fbPulseCtrl[1].Q;
fbPulseCtrl[1].RT;
fbPulseCtrl[2].Q;
fbPulseCtrl[2].RT;
fbPulseCtrl[3].Q;
fbPulseCtrl[3].RT;
fbPulseCtrl[4].Q;
fbPulseCtrl[4].RT;
fbPulseCtrl[5].Q;
fbPulseCtrl[5].RT;
fbPulseCtrl[6].Q;
fbPulseCtrl[6].RT;
fbPulseCtrl[7].Q;
fbPulseCtrl[7].RT;
fbPulseCtrl[8].Q;
fbPulseCtrl[8].RT;


IF bWaterOn AND ( bWaterOn2   OR    ABS( arrAxisCtrl[P1AxisNo.GMWind_U].Status.fActVelo)>=5 AND  ABS (arrAxisCtrl[P1AxisNo.GMWind_D].Status.fActVelo)>=5 )   THEN
  //P3EL2889S[3,5]:= fbPulseCtrl[9].Q;
   P1EL2889S[3,1]:= fbPulseCtrl[9].Q;
   P1EL2889S[3,2]:= fbPulseCtrl[9].Q;

   P2EL2889S[4,1]:=fbPulseCtrl[9].Q	;	
   P2EL2889S[4,2]:=fbPulseCtrl[9].Q;	

   P2EL2889S[4,3]:=fbPulseCtrl[9].Q	;	
   P2EL2889S[4,4]:=fbPulseCtrl[9].Q;	

ELSE
  //P3EL2889S[3,5]:= FALSE;
   P1EL2889S[3,1]:= FALSE;
   P1EL2889S[3,2]:= FALSE;
   P2EL2889S[4,1]:= FALSE	;	
   P2EL2889S[4,2]:= FALSE;	

   P2EL2889S[4,3]:=FALSE	;	
   P2EL2889S[4,4]:=FALSE;	
END_IF


//P1EL2889S[3,1]


*)
END_ACTION

ACTION TempBasic:


FOR i:=1 TO MaxTemp DO   //显示温度转换
	IF TempPVs[i].iPV1<>9999 THEN
		TempPVs[i].fPV1:=TempPVs[i].iPV1/10;	
	ELSE
		TempPVs[i].fPV1:=999.9;
	END_IF
    arrTempCtrl[i].fPVShow1:=TempPVs[i].fPV1;
	
	IF TempPVs[i].iPV2<>9999 THEN
		TempPVs[i].fPV2:=TempPVs[i].iPV2/10;
	ELSE
		TempPVs[i].fPV2:=999.9;
	END_IF
	 arrTempCtrl[i].fPVShow2:=TempPVs[i].fPV2;

	IF TempPVs[i].iPV3<>9999 THEN
		TempPVs[i].fPV3:=TempPVs[i].iPV3/10;
	ELSE
		TempPVs[i].fPV3:=999.9;
	END_IF
	 arrTempCtrl[i].fPVShow3:=TempPVs[i].fPV3;

	IF TempPVs[i].iPV4<>9999 THEN
		TempPVs[i].fPV4:=TempPVs[i].iPV4/10;
	ELSE
		TempPVs[i].fPV4:=999.9;
	END_IF
    arrTempCtrl[i].fPVShow4:=TempPVs[i].fPV4;
END_FOR

//温度控制
FOR i:=1 TO MaxTemp DO
     fbTemp[i](bReset:=P3_SystemRUN.bReset , ParTemp:=arrTempPar[i] , TempCtrl:=arrTempCtrl[i] );
END_FOR
END_ACTION

END_PROGRAM

// ---- P3POUs/P3FB/FB_Temperature.TcPOU
FUNCTION_BLOCK FB_Temperature    //温控功能块
VAR_INPUT
    bReset          :BOOL;
	ParTemp      : ST_ParTemperature;
END_VAR

VAR_IN_OUT
     TempCtrl:     STTempCtrl;
END_VAR
VAR_OUTPUT
    
END_VAR




VAR
       fTempMax                                :REAL;     //温度上限
      fTempMin                                 :REAL;     //温度下限


       rtTemp  :ARRAY[1..4] OF Tc2_Standard.R_TRIG;
	  iCountShow: INT;  //使用的显示通道数量
	  TemTON :Tc2_Standard.TON;
END_VAR

ParTemp.fTempArea:=5;
TemTON(PT:=T#300S);

TempCtrl.Tem_fPV:=TempCtrl.In.fPV-ParTemp.Tem_Offset;
TempCtrl.fPVShow_1:=TempCtrl.fPVShow1-ParTemp.Tem_Offset;
TempCtrl.In.fPV:=TempCtrl.In.iPV/10; //当前温度显示

TempCtrl.Out.iSV:=           REAL_TO_INT(ParTemp.fTempSet+ParTemp.Tem_Offset)*10; //控制温度设定值
//TempCtrl.Out.iPV_Offset:= REAL_TO_INT(ParTemp.fTempSet)*10;//控制温度设定值

//启动加热时候   如果当前温度到达设定温度 范围内则开始 判断温度超温和低温报警     
//启动加热5分钟  当前温度还未到达设定温度范围  则报警低温报警
//控制温度和显示温度实时检测差值并判断报警


(**自整定报警**)
TempCtrl.bTuningError:=TempCtrl.In.AutoTuningerr;  //
(**超温报警**)
//IF TempCtrl.In.AutoTuningON OR TempCtrl.In.HeatingON THEN
      rtTemp[1](CLK:=TempCtrl.Tem_fPV>ParTemp.fTempMax , Q=> );  //超温报警
      IF  (*rtTemp[1].Q*) TempCtrl.Tem_fPV>ParTemp.fTempMax+5 OR TempCtrl.fPVShow_1 >ParTemp.fTempMax+10 THEN
          TempCtrl.bTempError_HI:=TRUE;
      END_IF
//END_IF


(**传感器检测异常报警**)
  iCountShow:=SEL(TempCtrl.fPVShow_1<>999.9, 0,1)+SEL(TempCtrl.fPVShow2<>999.9, 0,1) +SEL(TempCtrl.fPVShow3<>999.9, 0,1) + SEL(TempCtrl.fPVShow4<>999.9, 0,1) ;

CASE  iCountShow OF 
1:
IF TempCtrl.In.PIDON AND  ABS (ParTemp.fTempSet-TempCtrl.Tem_fPV)<ParTemp.fTempArea AND NOT TempCtrl.bSenserError AND NOT TempCtrl.bTempError_HI  THEN
	iCountShow:=10;
END_IF

 
 
10:
    
      rtTemp[2](CLK:=ABS (TempCtrl.Tem_fPV-TempCtrl.fPVShow_1)>=ParTemp.fTempArea , Q=> );  //超温报警
       IF ABS (TempCtrl.Tem_fPV-TempCtrl.fPVShow_1)>=ParTemp.fTempArea THEN
             TempCtrl.bSenserError:=TRUE;
      END_IF
	  IF NOT TempCtrl.In.PIDON THEN
		  iCountShow:=0;
	  END_IF
	  
(*2:
      rtTemp[2](CLK:=ABS (TempCtrl.In.fPV-TempCtrl.fPVShow1)>=ParTemp.fTempArea  OR   
                              ABS (TempCtrl.In.fPV-TempCtrl.fPVShow2)>=ParTemp.fTempArea, Q=> );  //超温报警
       IF rtTemp[2].Q THEN
             TempCtrl.bSenserError:=TRUE;
      END_IF
3:
      rtTemp[2](CLK:=ABS (TempCtrl.In.fPV-TempCtrl.fPVShow1)>=ParTemp.fTempArea  OR   
                              ABS (TempCtrl.In.fPV-TempCtrl.fPVShow2)>=ParTemp.fTempArea  OR   
                              ABS (TempCtrl.In.fPV-TempCtrl.fPVShow3)>=ParTemp.fTempArea, Q=> );  //超温报警
       IF rtTemp[2].Q THEN
             TempCtrl.bSenserError:=TRUE;
      END_IF
4:
      rtTemp[2](CLK:=ABS (TempCtrl.In.fPV-TempCtrl.fPVShow1)>=ParTemp.fTempArea  OR   
                              ABS (TempCtrl.In.fPV-TempCtrl.fPVShow2)>=ParTemp.fTempArea  OR   
                              ABS (TempCtrl.In.fPV-TempCtrl.fPVShow3)>=ParTemp.fTempArea  OR   
                              ABS (TempCtrl.In.fPV-TempCtrl.fPVShow4)>=ParTemp.fTempArea, Q=> );  //超温报警
       IF rtTemp[2].Q THEN
             TempCtrl.bSenserError:=TRUE;
      END_IF*)
END_CASE

 IF TempCtrl.In.PIDON AND ABS (ParTemp.fTempSet-TempCtrl.Tem_fPV)>=ParTemp.fTempArea THEN
	 TemTON.IN:=TRUE;
	 ELSE
    TemTON.IN:=FALSE;	 
 END_IF
IF TemTON.Q THEN
	TempCtrl.bTempError_LI:=TRUE;
END_IF

IF bReset AND ( TempCtrl.bTempError_HI OR TempCtrl.bSenserError OR TempCtrl.bTempError_LI ) THEN
    TempCtrl.bTempError_HI:=FALSE;
    TempCtrl.bSenserError:=FALSE;
	TempCtrl.bTempError_LI:=FALSE;
END_IF


IF TempCtrl.bTempError_HI OR TempCtrl.bSenserError OR TempCtrl.bTempError_LI THEN
	TempCtrl.Out.PIDRun:=FALSE;
END_IF















(*
rtRec[1](CLK:=RecCtrl.Cmd.bLock , Q=> );
rtRec[2](CLK:=RecCtrl.Cmd.bAuto , Q=> );
rtRec[3](CLK:=RecCtrl.Cmd.bManual , Q=> );
rtRec[4](CLK:=RecCtrl.Cmd.bCentre , Q=> );

IF rtRec[1].Q   THEN  //外部锁定
    RecCtrl.Io.boLock:=TRUE;
    RecCtrl.Io.boAuto:=FALSE;
    RecCtrl.Io.boManual:=FALSE;
    RecCtrl.Io.boCentre:=FALSE;
END_IF

IF rtRec[2].Q   THEN  //自动
    RecCtrl.Io.boLock:=FALSE;
    RecCtrl.Io.boAuto:=TRUE;
    RecCtrl.Io.boManual:=FALSE;
    RecCtrl.Io.boCentre:=FALSE;
END_IF

IF rtRec[3].Q   THEN  //手动
    RecCtrl.Io.boLock:=FALSE;
    RecCtrl.Io.boAuto:=FALSE;
    RecCtrl.Io.boManual:=TRUE;
    RecCtrl.Io.boCentre:=FALSE;
END_IF

IF rtRec[4].Q   THEN  //居中
    RecCtrl.Io.boLock:=FALSE;
    RecCtrl.Io.boAuto:=FALSE;
    RecCtrl.Io.boManual:=FALSE;
    RecCtrl.Io.boCentre:=TRUE;
END_IF


RecCtrl.Status.bError:=RecCtrl.Io.biError;
RecCtrl.Status.bRuning:=RecCtrl.Io.biCentre;


*)

END_FUNCTION_BLOCK

// ---- P3POUs/POUs/Auxiliary/LateBlanking_Alarm.TcPOU
PROGRAM LateBlanking_Alarm
VAR
	Twinkle :ARRAY[1..20] OF FB_Blink;
	FB_Blink_11: FB_Blink;
	Alarm_TON :ARRAY[1..100] OF Tc2_Standard.TON;
	 AxisHandautomatic1: FB_AxisHandautomatic_1;
	 rAlarm :ARRAY[1..10] OF R_TRIG;
	 CleanTrig: R_TRIG;
END_VAR

QY_error:=YL_I[1];
Alarm();

Alarm_TON[1](PT:=T#5S);
Alarm_TON[2](PT:=T#5S);
Alarm_TON[3](PT:=T#5S);
Alarm_TON[4](PT:=T#8S);
Alarm_TON[5](PT:=T#8S);
Alarm_TON[6](PT:=T#10MS);
Alarm_TON[7](PT:=T#10MS);
Alarm_TON[8](PT:=T#10MS);
Alarm_TON[9](PT:=T#10MS);
Alarm_TON[10](PT:=T#10MS);
Alarm_TON[11](PT:=T#10MS);
Alarm_TON[12](PT:=T#10MS);
Alarm_TON[13](PT:=T#10MS);
Alarm_TON[14](PT:=T#10MS);
Alarm_TON[15](PT:=T#100MS);
Alarm_TON[16](PT:=T#100MS);
Alarm_TON[17](PT:=T#100MS);
Alarm_TON[18](PT:=T#100MS);
Alarm_TON[19](PT:=T#20MS);
Alarm_TON[20](PT:=T#6S);
Alarm_TON[25](PT:=T#60MS);
Alarm_TON[26](PT:=T#60MS);
Alarm_TON[27](PT:=T#200MS);
Alarm_TON[31](PT:=T#1.1S);
Alarm_TON[32](PT:=T#1.1S);
Alarm_TON[33](PT:=T#1.1S);
Alarm_TON[34](PT:=T#1000MS);
Alarm_TON[35](PT:=T#2000MS);
Alarm_TON[36](PT:=T#2S);
Alarm_TON[37](PT:=T#2S);
Alarm_TON[38](PT:=T#60MS);
Alarm_TON[39](PT:=T#60MS);
Alarm_TON[40](PT:=T#3S);
//尾段报警总结
IF  arrAxisCtrl[P3AxisNo.P3M1_ColdpreActuated].Status.Error             OR arrAxisCtrl[P3AxisNo.P3M1_ColdpreLine].Status.Error           OR
	arrAxisCtrl[P3AxisNo.P3M1_ColdpreRetracting].Status.Error           OR arrAxisCtrl[P3AxisNo.P3M1_ColdpreSupPlateLine].Status.Error   OR
	arrAxisCtrl[P3AxisNo.P3M1_ColdpreUpDown].Status.Error               OR arrAxisCtrl[P3AxisNo.P3M1_ColdpreWhirling].Status.Error       OR
	arrAxisCtrlV2[P3AxisNo.P3_M2_OvenCarrying].Status.Error             OR arrAxisCtrlV2[P3AxisNo.P3_M2_OvenRetracting].Status.Error       OR
	arrAxisCtrlV2[P3AxisNo.P3_M2_OvenUpDown].Status.Error               OR arrAxisCtrl[P3AxisNo.P3_M3_HotPressingActuated].Status.Error  OR
	arrAxisCtrl[P3AxisNo.P3_M3_HotPressingLine].Status.Error            OR arrAxisCtrl[P3AxisNo.P3_M4_OffloadingCarrying].Status.Error   OR
	arrAxisCtrl[P3AxisNo.P3_M4_OffloadingUpDown].Status.Error           OR arrAxisCtrl[P3AxisNo.P3_M4_SortingoutCarrying].Status.Error   OR
	//arrAxisCtrl[P3AxisNo.P3_M4_SortingoutUpDown].Status.Error           OR arrAxisCtrl[P3AxisNo.P3_M4_WeighLine].Status.Error            OR
	arrAxisCtrl[P3AxisNo.P3_M4_WeighUpDown].Status.Error                OR arrAxisCtrl[P3AxisNo.P3_M4_WeighWhirling].Status.Error        OR
	//一号叠台、尾卷、贴胶电机报警
	
	(*arrCyCtrl[P3CYNo.P3ColdPressClip].Status.Error1                     OR*) (*arrCyCtrl[P3CYNo.P3ColdPressTensed].Status.Error1             OR
	arrCyCtrl[P3CYNo.P3HotPressTensed].Status.Error1                    OR*arrCyCtrl[P3CYNo.P3OvenMoveClip].Status.Error1           (  OR
	arrCyCtrl[P3CYNo.P3ShortTest].Status.Error1                        OR*)  arrCyCtrl[P3CYNo.P3SortClamp].Status.Error1                   OR
	arrCyCtrl[P3CYNo.P3SortLifting].Status.Error1                       OR arrCyCtrl[P3CYNo.P3SortRotate].Status.Error1                  OR
	arrCyCtrl[P3CYNo.P3ThicknessMeasuringSwitch].Status.Error1          OR arrCyCtrl[P3CYNo.P3ThicknessPressure].Status.Error1           OR
	arrCyCtrl[P3CYNo.P3ThicknessSupport].Status.Error1                  OR arrCyCtrl[P3CYNo.P3WeightFeedingClamp].Status.Error1          OR
	arrCyCtrl[P3CYNo.P3BoxLock1_NG].Status.Error1                       OR arrCyCtrl[P3CYNo.P3BoxLock2_NG].Status.Error1                 OR
	arrCyCtrl[P3CYNo.P3BoxLock3_NG].Status.Error1                       OR arrCyCtrl[P3CYNo.P3BlankingClamp].Status.Error1               OR
	arrCyCtrl[P3CYNo.P3BlankingLifting].Status.Error1                   OR arrCyCtrl[P3CYNo.P3Oven1].Status.Error1                       OR
	arrCyCtrl[P3CYNo.P3Oven2].Status.Error1                             OR arrCyCtrl[P3CYNo.P3Oven3].Status.Error1                       OR
	arrCyCtrl[P3CYNo.P3Oven4].Status.Error1                             OR arrCyCtrl[P3CYNo.P3Oven5].Status.Error1                       OR
	arrCyCtrl[P3CYNo.P3Oven6].Status.Error1                             OR arrCyCtrl[P3CYNo.P3Oven7].Status.Error1                       OR
	arrCyCtrl[P3CYNo.P3Oven8].Status.Error1                             OR arrCyCtrl[P3CYNo.P3Oven9].Status.Error1                       OR
	arrCyCtrl[P3CYNo.P3Oven10].Status.Error1                            OR arrCyCtrl[P3CYNo.P3Oven11].Status.Error1                      OR
	arrCyCtrl[P3CYNo.P3Oven12].Status.Error1                            OR arrCyCtrl[P3CYNo.P3Oven13].Status.Error1                      OR
	arrCyCtrl[P3CYNo.P3Oven14].Status.Error1                            OR arrCyCtrl[P3CYNo.P3Oven15].Status.Error1                      OR
	arrCyCtrl[P3CYNo.P3Oven16].Status.Error1                            OR arrCyCtrl[P3CYNo.P3Oven17].Status.Error1                      OR
	arrCyCtrl[P3CYNo.P3Oven18].Status.Error1                            OR arrCyCtrl[P3CYNo.P3Oven19].Status.Error1                      OR
	arrCyCtrl[P3CYNo.P3Oven20].Status.Error1                            OR arrCyCtrl[P3CYNo.P3Oven21].Status.Error1                      OR
	arrCyCtrl[P3CYNo.P3CellPush].Status.Error1                          OR arrCyCtrl[P3CYNo.P3CellAdvance].Status.Error1                 OR
	arrCyCtrl[P3CYNo.P3TapePush].Status.Error1                          OR arrCyCtrl[P3CYNo.P3TapePull].Status.Error1                    OR
	arrCyCtrl[P3CYNo.P3TapeLift].Status.Error1                          OR arrCyCtrl[P3CYNo.P3TapeCut].Status.Error1                     OR
	arrCyCtrl[P3CYNo.P3GluePush].Status.Error1                          OR arrCyCtrl[P3CYNo.P3TapeBuffer].Status.Error1                  OR
	arrCyCtrl[P3CYNo.P3TapeSpin].Status.Error1                          OR arrCyCtrl[P3CYNo.P3WgightUP].Status.Error1                    OR
	arrCyCtrl[P3CYNo.P3SortPush].Status.Error1                          OR arrCyCtrl[P3CYNo.P3CellPushSpin].Status.Error1                OR
	arrCyCtrl[P3CYNo.P3CellSpin].Status.Error1                          OR arrCyCtrl[P3CYNo.P3_GlueExtend].Status.Error1                 OR
	arrCyCtrl[P3CYNo.P3_GluePress].Status.Error1                        OR arrCyCtrl[P3CYNo.P3_GlueCut].Status.Error1                    OR
	arrCyCtrl[P3CYNo.P3_GluePull].Status.Error1                         OR
    //尾段气缸ON报警
	
	arrCyCtrl[P3CYNo.P3ColdPressClip].Status.Error2                     OR (*arrCyCtrl[P3CYNo.P3ColdPressTensed].Status.Error2             OR
	arrCyCtrl[P3CYNo.P3HotPressTensed].Status.Error2                    OR*) arrCyCtrl[P3CYNo.P3OvenMoveClip].Status.Error2              OR
	arrCyCtrl[P3CYNo.P3ShortTest].Status.Error2                         OR arrCyCtrl[P3CYNo.P3SortClamp].Status.Error2                   OR
	(*arrCyCtrl[P3CYNo.P3SortLifting].Status.Error2                       OR *)arrCyCtrl[P3CYNo.P3SortRotate].Status.Error2              OR
	arrCyCtrl[P3CYNo.P3ThicknessMeasuringSwitch].Status.Error2          OR arrCyCtrl[P3CYNo.P3ThicknessPressure].Status.Error2           OR
	arrCyCtrl[P3CYNo.P3ThicknessSupport].Status.Error2                  OR(* arrCyCtrl[P3CYNo.P3WeightFeedingClamp].Status.Error2          OR*)
	arrCyCtrl[P3CYNo.P3BoxLock1_NG].Status.Error2                       OR arrCyCtrl[P3CYNo.P3BoxLock2_NG].Status.Error2                 OR
	arrCyCtrl[P3CYNo.P3BoxLock3_NG].Status.Error2                       OR arrCyCtrl[P3CYNo.P3BlankingClamp].Status.Error2               OR
	arrCyCtrl[P3CYNo.P3BlankingLifting].Status.Error2                   OR arrCyCtrl[P3CYNo.P3Oven1].Status.Error2                       OR
	arrCyCtrl[P3CYNo.P3Oven2].Status.Error2                             OR arrCyCtrl[P3CYNo.P3Oven3].Status.Error2                       OR
	arrCyCtrl[P3CYNo.P3Oven4].Status.Error2                             OR arrCyCtrl[P3CYNo.P3Oven5].Status.Error2                       OR
	arrCyCtrl[P3CYNo.P3Oven6].Status.Error2                             OR arrCyCtrl[P3CYNo.P3Oven7].Status.Error2                       OR
	arrCyCtrl[P3CYNo.P3Oven8].Status.Error2                             OR arrCyCtrl[P3CYNo.P3Oven9].Status.Error2                       OR
	arrCyCtrl[P3CYNo.P3Oven10].Status.Error2                            OR arrCyCtrl[P3CYNo.P3Oven11].Status.Error2                      OR
	arrCyCtrl[P3CYNo.P3Oven12].Status.Error2                            OR arrCyCtrl[P3CYNo.P3Oven13].Status.Error2                      OR
	arrCyCtrl[P3CYNo.P3Oven14].Status.Error2                            OR arrCyCtrl[P3CYNo.P3Oven15].Status.Error2                      OR
	arrCyCtrl[P3CYNo.P3Oven16].Status.Error2                            OR arrCyCtrl[P3CYNo.P3Oven17].Status.Error2                      OR
	arrCyCtrl[P3CYNo.P3Oven18].Status.Error2                            OR arrCyCtrl[P3CYNo.P3Oven19].Status.Error2                      OR
	arrCyCtrl[P3CYNo.P3Oven20].Status.Error2                            OR arrCyCtrl[P3CYNo.P3Oven21].Status.Error2                      OR
	arrCyCtrl[P3CYNo.P3CellPush].Status.Error2                          OR arrCyCtrl[P3CYNo.P3CellAdvance].Status.Error2                 OR
	arrCyCtrl[P3CYNo.P3TapePush].Status.Error2                          OR arrCyCtrl[P3CYNo.P3TapePull].Status.Error2                    OR
	arrCyCtrl[P3CYNo.P3TapeLift].Status.Error2                          OR arrCyCtrl[P3CYNo.P3TapeCut].Status.Error2                     OR
	arrCyCtrl[P3CYNo.P3GluePush].Status.Error2                          OR arrCyCtrl[P3CYNo.P3TapeBuffer].Status.Error2                  OR
	arrCyCtrl[P3CYNo.P3TapeSpin].Status.Error2                          OR arrCyCtrl[P3CYNo.P3WgightUP].Status.Error2                    OR
	arrCyCtrl[P3CYNo.P3SortPush].Status.Error2                          OR arrCyCtrl[P3CYNo.P3CellPushSpin].Status.Error2                OR
	arrCyCtrl[P3CYNo.P3CellSpin].Status.Error2                         (* OR arrCyCtrl[P3CYNo.P3_GlueExtend].Status.Error2         *)        OR
	arrCyCtrl[P3CYNo.P3_GluePress].Status.Error2                        OR arrCyCtrl[P3CYNo.P3_GlueCut].Status.Error2                    OR
	arrCyCtrl[P3CYNo.P3_GluePull].Status.Error2                         OR
 
    //尾段气缸OFF报警
   
	arrTempCtrl[1].bSenserError                                         OR arrTempCtrl[1].bTempError_HI                                  OR
	arrTempCtrl[2].bSenserError                                         OR arrTempCtrl[2].bTempError_HI                                  OR
	arrTempCtrl[3].bSenserError                                         OR arrTempCtrl[3].bTempError_HI                                  OR
	arrTempCtrl[4].bSenserError                                         OR arrTempCtrl[4].bTempError_HI                                  OR
	arrTempCtrl[5].bSenserError                                         OR arrTempCtrl[5].bTempError_HI                                  OR
	arrTempCtrl[6].bSenserError                                         OR arrTempCtrl[6].bTempError_HI                                  OR
	arrTempCtrl[7].bSenserError                                         OR arrTempCtrl[7].bTempError_HI                                  OR
	arrTempCtrl[8].bSenserError                                         OR arrTempCtrl[8].bTempError_HI                                  OR
	arrTempCtrl[9].bSenserError                                         OR arrTempCtrl[9].bTempError_HI                                  OR
	arrTempCtrl[10].bSenserError                                        OR arrTempCtrl[10].bTempError_HI                                 OR
	arrTempCtrl[11].bSenserError                                        OR arrTempCtrl[11].bTempError_HI                                 OR
	arrTempCtrl[12].bSenserError                                        OR arrTempCtrl[12].bTempError_HI                                 OR
	arrTempCtrl[13].bSenserError                                        OR arrTempCtrl[13].bTempError_HI                                 OR
	arrTempCtrl[14].bSenserError                                        OR arrTempCtrl[14].bTempError_HI                                 OR
	arrTempCtrl[15].bSenserError                                        OR arrTempCtrl[15].bTempError_HI                                 OR
	arrTempCtrl[16].bSenserError                                        OR arrTempCtrl[16].bTempError_HI                                 OR
	arrTempCtrl[17].bSenserError                                        OR arrTempCtrl[17].bTempError_HI                                 OR
	arrTempCtrl[18].bSenserError                                        OR arrTempCtrl[18].bTempError_HI                                 OR
	arrTempCtrl[19].bSenserError                                        OR arrTempCtrl[19].bTempError_HI                                 OR
	arrTempCtrl[20].bSenserError                                        OR arrTempCtrl[20].bTempError_HI                                 OR
	arrTempCtrl[21].bSenserError                                        OR arrTempCtrl[21].bTempError_HI                                 OR
	arrTempCtrl[22].bSenserError                                        OR arrTempCtrl[22].bTempError_HI                                 OR
	arrTempCtrl[23].bSenserError                                        OR arrTempCtrl[23].bTempError_HI                                 OR
	arrTempCtrl[24].bSenserError                                        OR arrTempCtrl[24].bTempError_HI                                 OR
	arrTempCtrl[25].bSenserError                                        OR arrTempCtrl[25].bTempError_HI                                 OR
	arrTempCtrl[26].bSenserError                                        OR arrTempCtrl[26].bTempError_HI                                 OR
	arrTempCtrl[27].bSenserError                                        OR arrTempCtrl[27].bTempError_HI                                 OR
	arrTempCtrl[28].bSenserError                                        OR arrTempCtrl[28].bTempError_HI                                 OR
	arrTempCtrl[29].bSenserError                                        (*OR arrTempCtrl[29].bTempError_HI*)                                 OR
	arrTempCtrl[30].bSenserError                                       (* OR arrTempCtrl[30].bTempError_HI *)                                OR
	arrTempCtrl[31].bSenserError                                       (* OR arrTempCtrl[31].bTempError_HI*)                                 OR
	arrTempCtrl[32].bSenserError                                       (* OR arrTempCtrl[32].bTempError_HI*)                                 OR
	arrTempCtrl[33].bSenserError                                        OR arrTempCtrl[33].bTempError_HI                                 OR
	arrTempCtrl[34].bSenserError                                        OR arrTempCtrl[34].bTempError_HI                                 OR
	arrTempCtrl[35].bSenserError                                        OR arrTempCtrl[35].bTempError_HI                                 OR
	arrTempCtrl[36].bSenserError                                        OR arrTempCtrl[36].bTempError_HI                                 OR
	arrTempCtrl[37].bSenserError                                        OR arrTempCtrl[37].bTempError_HI                                 OR
	arrTempCtrl[38].bSenserError                                        OR arrTempCtrl[38].bTempError_HI                                 OR
	arrTempCtrl[39].bSenserError                                        OR arrTempCtrl[39].bTempError_HI                                 OR
	arrTempCtrl[40].bSenserError                                        OR arrTempCtrl[40].bTempError_HI                                 OR
	arrTempCtrl[41].bSenserError                                        OR arrTempCtrl[41].bTempError_HI                                 OR
	arrTempCtrl[42].bSenserError                                        OR arrTempCtrl[42].bTempError_HI                                 OR
	arrTempCtrl[43].bSenserError                                        OR arrTempCtrl[43].bTempError_HI                                 OR
	arrTempCtrl[44].bSenserError                                        OR arrTempCtrl[44].bTempError_HI                                 OR
	arrTempCtrl[45].bSenserError                                        OR arrTempCtrl[45].bTempError_HI                                 OR
	arrTempCtrl[46].bSenserError                                        OR arrTempCtrl[46].bTempError_HI                                 OR
	arrTempCtrl[47].bSenserError                                        OR arrTempCtrl[47].bTempError_HI                                 OR
	arrTempCtrl[48].bSenserError                                        OR arrTempCtrl[48].bTempError_HI                                 OR
	arrTempCtrl[49].bSenserError                                        OR arrTempCtrl[49].bTempError_HI                                 OR
	arrTempCtrl[50].bSenserError                                        OR arrTempCtrl[50].bTempError_HI                                 OR
	arrTempCtrl[51].bSenserError                                        OR arrTempCtrl[51].bTempError_HI                                 OR
	arrTempCtrl[52].bSenserError                                        OR arrTempCtrl[52].bTempError_HI                                 OR
	arrTempCtrl[53].bSenserError                                        OR arrTempCtrl[53].bTempError_HI                                 OR
	arrTempCtrl[54].bSenserError                                        OR arrTempCtrl[54].bTempError_HI                                 OR
	arrTempCtrl[55].bSenserError                                        OR arrTempCtrl[55].bTempError_HI                                 OR
	arrTempCtrl[56].bSenserError                                        OR arrTempCtrl[56].bTempError_HI                                 OR
	arrTempCtrl[57].bSenserError                                        OR arrTempCtrl[57].bTempError_HI                                 OR
	arrTempCtrl[58].bSenserError                                        OR arrTempCtrl[58].bTempError_HI                                 OR
	arrTempCtrl[59].bSenserError                                        OR arrTempCtrl[59].bTempError_HI                                 OR
	arrTempCtrl[60].bSenserError                                        OR arrTempCtrl[50].bTempError_HI                                 OR
	arrTempCtrl[61].bSenserError                                        OR arrTempCtrl[51].bTempError_HI                                 OR
	arrTempCtrl[62].bSenserError                                        OR arrTempCtrl[52].bTempError_HI                                 OR
	arrTempCtrl[63].bSenserError                                        OR arrTempCtrl[53].bTempError_HI                                 OR
	arrTempCtrl[64].bSenserError                                        OR arrTempCtrl[54].bTempError_HI                                 OR
	arrTempCtrl[65].bSenserError                                        OR arrTempCtrl[55].bTempError_HI                                 OR
	arrTempCtrl[66].bSenserError                                        OR arrTempCtrl[56].bTempError_HI                                 OR
	arrTempCtrl[67].bSenserError                                        OR arrTempCtrl[57].bTempError_HI                                 OR
	arrTempCtrl[68].bSenserError                                        OR arrTempCtrl[58].bTempError_HI                                 OR
	arrTempCtrl[69].bSenserError                                        OR arrTempCtrl[69].bTempError_HI                                 OR
	arrTempCtrl[70].bSenserError                                        OR arrTempCtrl[70].bTempError_HI                                 OR
	arrTempCtrl[71].bSenserError                                        OR arrTempCtrl[71].bTempError_HI                                 OR
	arrTempCtrl[72].bSenserError                                        OR arrTempCtrl[72].bTempError_HI                                 OR
	arrTempCtrl[73].bSenserError                                        OR arrTempCtrl[73].bTempError_HI                                 OR
	arrTempCtrl[74].bSenserError                                        OR arrTempCtrl[74].bTempError_HI                                 OR
	arrTempCtrl[75].bSenserError                                        OR arrTempCtrl[75].bTempError_HI                                 OR
	arrTempCtrl[76].bSenserError                                        OR arrTempCtrl[76].bTempError_HI                                 OR
	arrTempCtrl[77].bSenserError                                        OR arrTempCtrl[77].bTempError_HI                                 OR
	arrTempCtrl[78].bSenserError                                        OR arrTempCtrl[78].bTempError_HI                                 OR
	arrTempCtrl[79].bSenserError                                        OR arrTempCtrl[79].bTempError_HI                                 OR
	arrTempCtrl[80].bSenserError                                        OR arrTempCtrl[80].bTempError_HI                                 OR
	arrTempCtrl[81].bSenserError                                        OR arrTempCtrl[81].bTempError_HI                                 OR
	arrTempCtrl[82].bSenserError                                        OR arrTempCtrl[82].bTempError_HI                                 OR
	arrTempCtrl[83].bSenserError                                        OR arrTempCtrl[83].bTempError_HI                                 OR
	arrTempCtrl[84].bSenserError                                        OR arrTempCtrl[84].bTempError_HI                                 OR
	arrTempCtrl[85].bSenserError                                        OR arrTempCtrl[85].bTempError_HI                                 OR
	arrTempCtrl[86].bSenserError                                        OR arrTempCtrl[86].bTempError_HI                                 OR
	P3_Error[1]															OR P3_Error[2]										     		 OR 
	P3_Error[3]															OR P3_Error[4]										     		 OR 
	P3_Error[5]															OR P3_Error[6]										     		 OR 
  (*P3_Error[7]  														OR P3_Error[8]										     		 OR*)  
	P3_Error[9]															OR P3_Error[10]										     		 OR 
	P3_Error[11]														OR P3_Error[12]										     		 OR 
	(*P3_Error[13]														OR*) P3_Error[14]										     	 OR  
	P3_Error[15]														OR P3_Error[16]										     		 OR 
	P3_Error[17]														OR P3_Error[18]										     		 OR
	P3_Error[19]														OR P3_Error[20]										     		 OR 
	P3_Error[21]														OR P3_Error[22]										     		 OR  
	P3_Error[23]														OR P3_Error[24]										     		 OR 
	P3_Error[25]														(*OR P3_Error[26]										     	*)	 OR   
	P3_Error[27]														OR P3_Error[28]										     		 OR 
	P3_Error[29]														OR P3_Error[30]										     		 OR  
	P3_Error[31]														OR P3_Error[32]										     		 OR 
	P3_Error[33]														OR P3_Error[34]										     		 OR
	P3_Error[35]														OR P3_Error[36]										     		 OR 
	P3_Error[37]														OR P3_Error[38]										     		 OR  
	P3_Error[39]														OR P3_Error[40]												OR
 	P3_Error[42]														OR P3_Error[45]												 OR 
	P3_Error[46]														OR P3_Error[47]												 OR 
	P3_Error[48]														OR P3_Error[50]									                 	OR 
	P3_Error[53]														OR P3_Error[54]												OR
	P3_Error[57]														OR P3_Error[58]												OR
	P3_Error[59]														OR P3_Error[60]												OR
	P3_Error[61]														OR P3_Error[62]												OR
	P3_Error[63]														OR P3_Error[64]												OR
	P3_Error[65]														OR P3_Error[66]												OR
	P3_Error[67]														OR P3_Error[68]												OR	
	P3_Error[69]														OR P3_Error[70]											OR
	P3_Error[71]														OR P3_Error[72]											OR	
	P3_Error[73]														OR P3_Error[74]														OR 
	P3_Error[75]														OR P3_Error[79]													OR 
	P3_Error[87]														OR P3_Error[89]											OR 
	P3_Error[93]                                                        OR
	P3_Error[120]														OR P3_Error[121]										OR 
	P3_Error[122]														OR P3_Error[123]										OR 
	P3_Error[124]														OR P3_Error[125]										OR 
	P3_Error[126]														OR P3_Error[127]										OR 
	Door_error[1]   		 											OR Door_error[2]												 OR
	Door_error[1]   		 											OR Door_error[2]												 OR
	Door_error[1]   		 											OR Door_error[2]												 OR
	Door_error[3]   		 											OR Door_error[4]												 OR
	Door_error[5]   		 											OR Door_error[6]												 OR
	Door_error[7]   		 											OR Door_error[8]												 OR
	Door_error[9]   		 											OR Door_error[10]												 OR
	Door_error[11]   		 											OR Door_error[12]												 OR
	Door_error[13]   		 											OR Door_error[14]												 OR
	Door_error[15]   		 											OR Door_error[16]												 OR
	bCodeConError														OR bCodeError													 OR
	P3_Tem_Error[1]														OR P3_Tem_Error[2]	                                             OR
	P3_Tem_Error[3]														OR P3_Tem_Error[4]	                                             OR
	P3_Tem_Error[5]														OR P3_Tem_Error[6]	                                             OR
	P3_Tem_Error[7]														OR P3_Tem_Error[8]	                                             OR
 	P3_Tem_Error[9]														OR P3_Tem_Error[10]	                                             OR
	P3_Tem_Error[11]													OR P3_Tem_Error[12]	                                             OR
	P3_Tem_Error[13]													OR P3_Tem_Error[14]	                                             OR
	P3_Tem_Error[15]													OR P3_Tem_Error[16]	                                             OR
	P3_Tem_Error[17]													OR P3_Tem_Error[18]	                                             OR
	P3_Tem_Error[19]													OR P3_Tem_Error[20]	                                             OR
	P3_Tem_Error[21]													OR P3_Tem_Error[22]	                                             OR
	P3_Tem_Error[23]													OR P3_Tem_Error[24]	                                             OR
	P3_Tem_Error[25]													OR P3_Tem_Error[26]	                                             OR
	P3_Tem_Error[27]													OR P3_Tem_Error[28]	                                             OR
	P3_Tem_Error[29]													OR P3_Tem_Error[30]	                                             OR
	P3_Tem_Error[31]													OR P3_Tem_Error[32]	                                             OR
	P3_Tem_Error[33]													OR P3_Tem_Error[34]	                                             OR
	P3_Tem_Error[35]													OR P3_Tem_Error[36]	                                             OR
	P3_Tem_Error[37]													OR P3_Tem_Error[38]	                                             OR
	P3_Tem_Error[39]													OR P3_Tem_Error[40]	                                             OR
	P3_Tem_Error[41]													OR P3_Tem_Error[42]	                                             OR
	P3_Tem_Error[43]													OR P3_Tem_Error[44]	                                             OR
	P3_Tem_Error[45]													OR P3_Tem_Error[46]	                                             OR
	P3_Tem_Error[47]													OR P3_Tem_Error[48]	                                             OR	
	P3_Tem_Error[49]													OR P3_Tem_Error[50]	                                             OR	
	P3_Tem_Error[51]													OR P3_Tem_Error[52]	                                             OR	
	P3_Tem_Error[53]													OR P3_Tem_Error[54]	                                             OR	
	P3_Tem_Error[55]													OR P3_Tem_Error[56]	                                             OR	
	P3_Tem_Error[57]													OR P3_Tem_Error[58]	                                             OR	
	P3_Tem_Error[59]													OR P3_Tem_Error[60]	                                             OR	
	P3_Tem_Error[61]													OR P3_Tem_Error[62]	                                             OR	
	P3_Tem_Error[63]													OR P3_Tem_Error[64]	                                             OR	
	P3_Tem_Error[65]													OR P3_Tem_Error[66]	                                             OR	
	P3_Tem_Error[67]													OR P3_Tem_Error[68]	                                             OR	
	P3_Tem_Error[69]													OR P3_Tem_Error[70]	                                             OR	
	P3_Tem_Error[71]													OR P3_Tem_Error[72]	                                             OR	
	P3_Tem_Error[73]													OR P3_Tem_Error[74]	                                             OR	
	P3_Tem_Error[75]													OR P3_Tem_Error[76]	                                             OR	
	P3_Tem_Error[77]													OR P3_Tem_Error[78]	                                             OR	
	P3_Tem_Error[79]													OR P3_Tem_Error[80]	                                             OR	
	P3_Tem_Error[81]													OR P3_Tem_Error[82]	                                             OR	
	P3_Tem_Error[83]													OR P3_Tem_Error[84]	                                             OR	
	P3_Tem_Error[85]													OR P3_Tem_Error[86]	                                             OR	
	P3_Tem_Error[87]													OR P3_Tem_Error[88]	                                             OR
	P3_Tem_Error[89]													OR P3_Tem_Error[90]	                                             OR
	P3_Tem_Error[91]													OR P3_Tem_Error[92]	                                             OR
	P3_Tem_Error[93]													OR P3_Tem_Error[94]	                                             OR
	P3_Tem_Error[95]													OR P3_Tem_Error[96]	                                             OR
 	QY_error 	                                                        OR P3Press.Pressure_Alarm[1]                                     OR						                                         
	P3Press.Pressure_Alarm[2] 
//扭矩报警
	OR HMI_TorAlarm_D[160]//冷呀上料夹平移力矩超限报警					
	OR HMI_TorAlarm_D[161]//冷压上料夹进退力矩超限报警
	OR HMI_TorAlarm_D[162]//冷压上料夹旋转力矩超限报警
	OR HMI_TorAlarm_D[165]//冷压驱动力矩超限报警
	OR HMI_TorAlarm_D[166]//烤箱上料夹搬运力矩超限报警
	OR HMI_TorAlarm_D[167]//烤箱上料夹进退力矩超限报警
	OR HMI_TorAlarm_D[170]//热压驱动力矩超限报警
	OR HMI_TorAlarm_D[171]//称重上料夹平移力矩超限报警
	OR HMI_TorAlarm_D[173]//称重上料夹旋转力矩超限报警
	OR HMI_TorAlarm_D[174]//电芯分选夹搬运力矩超限报警
	OR HMI_TorAlarm_D[176]//电芯下料夹搬运力矩超限报警
	OR P3_Error[42]
	OR AxisHandautomatic1.error
	OR P3_Error[86]
	//叠片冷压上料门禁
	OR NOT P2Senser.P2M1_Securitydoorswitch3 OR NOT P2Senser.P2M1_Securitydoorswitch4
	OR NOT P2Senser.P2M2_Securitydoorswitch3 OR NOT P2Senser.P2M2_Securitydoorswitch4
	OR NOT P2Senser.P2M3_Securitydoorswitch3 OR NOT P2Senser.P2M3_Securitydoorswitch4
	THEN
	
//烤箱及热压的温度报警
	
    b_Alarm[4]:=TRUE;		
END_IF

IF  b_Alarm[4] THEN
	P3_SystemRUN.btnAuto:=FALSE;
	P3_SystemRUN.hmiAuto:=FALSE;
END_IF

	IF b_Alarm[4] OR  P3_Error[42] THEN
		P3Senser.P3_Tricolorlamp_Red:=TRUE;
		P3Senser.P3_Tricolorlamp_Yellow:=FALSE;
		P3Senser.P3_Tricolorlamp_Green:=FALSE;
	ELSIF P3_SystemRUN.iMode=3 THEN
		P3Senser.P3_Tricolorlamp_Red:=FALSE;
		P3Senser.P3_Tricolorlamp_Yellow:=TRUE;
		P3Senser.P3_Tricolorlamp_Green:=FALSE;	
	ELSIF P3_SystemRUN.iMode=1 THEN
		P3Senser.P3_Tricolorlamp_Red:=FALSE;
		P3Senser.P3_Tricolorlamp_Yellow:=FALSE;
		P3Senser.P3_Tricolorlamp_Green:=TRUE;
	END_IF

// 热压有功能屏蔽报警
IF NOT P3User2_Par.Shield[5] AND (Mes1.Error[26] OR Mes1.Error[27] OR Mes1.Error[28] OR Mes1.Error[29] ) THEN	
	P3_Error[86]:=TRUE ;// 热压有功能屏蔽报警
END_IF	
	
//上位机未连接
IF NOT PC_heart AND NOT P3User2_Par.Shield[5] THEN
	IF NOT Alarm_TON[1].Q THEN
		Alarm_TON[1].IN:=TRUE;
	ELSE
			P3_Error[2]:=TRUE;//上位机未连接
	END_IF
ELSE
		Alarm_TON[1].IN:=FALSE;
END_IF

IF  PC_heart AND NOT P3User2_Par.Shield[5] THEN
	IF NOT Alarm_TON[2].Q THEN
		Alarm_TON[2].IN:=TRUE;
	ELSE
			P3_Error[2]:=TRUE;//上位机未连接
	END_IF
ELSE
		Alarm_TON[2].IN:=FALSE;
END_IF	

IF  (Step32=1077 AND NOT PC_finish1) AND NOT P3User2_Par.Shield[5] THEN
	IF NOT Alarm_TON[3].Q THEN
		Alarm_TON[3].IN:=TRUE;
	ELSE
		Step32:=1076;
		P3_Error[3]:=TRUE;//上位机上传叠片数据超时报警
	END_IF
ELSE
		Alarm_TON[3].IN:=FALSE;
END_IF

IF  (Step32=118 AND NOT Cold_finish) AND NOT P3User2_Par.Shield[5]  THEN
	IF NOT Alarm_TON[4].Q THEN
		Alarm_TON[4].IN:=TRUE;
	ELSE
			P3_Error[4]:=TRUE;//上位机校对数据超时报警
	END_IF
ELSE
		Alarm_TON[4].IN:=FALSE;
END_IF

IF  (Step35=198 AND NOT PC_finish) AND NOT P3User2_Par.Shield[5] THEN
	IF NOT Alarm_TON[5].Q THEN
		Alarm_TON[5].IN:=TRUE;
	ELSE
			P3_Error[5]:=TRUE;//上位机上传热压数据超时报警
	END_IF
ELSE
		Alarm_TON[5].IN:=FALSE;
END_IF


IF  PC_alarm[1] AND NOT P3User2_Par.Shield[5] THEN
	IF NOT Alarm_TON[6].Q THEN
		Alarm_TON[6].IN:=TRUE;
	ELSE
			P3_Error[6]:=TRUE;//物料已经用完,请更换上位机物料批次
			PC_alarm[1]:=FALSE;
	END_IF
ELSE
		Alarm_TON[6].IN:=FALSE;
END_IF
//////////////////////////////////////////////////////不良电芯总结//////////////////////////////////////////////////////////////////////////
rAlarm[1](CLK:=CellMemory[CellNo.Thickness].ScanCode<>1 AND CellMemory[CellNo.Thickness].Cell  AND Thickness_Finish AND Step35>=3000 AND Step35<3050   AND NOT P3User2_Par.Shield[4]  , Q=> );
IF rAlarm[1].Q THEN
	P3_Error[7]:=TRUE;//出料后,该电芯是扫码NG
END_IF

IF (NOT CellMemory[CellNo.Thickness].Cell_cold_result OR NOT CellMemory[CellNo.Thickness].Cell_cold_result1 OR NOT CellMemory[CellNo.Thickness].Cell_cold_result2)  AND Thickness_Finish  
AND CellMemory[CellNo.Thickness].Cell AND Step35>=3000 AND Step35<3050 AND CellMemory[CellNo.Thickness].ScanCode=1 
AND CellMemory[CellNo.Thickness].Hough=1 AND NOT P3User2_Par.Shield[4]  THEN
	IF NOT Alarm_TON[14].Q THEN
		Alarm_TON[14].IN:=TRUE;
	ELSE
		P3_Error[8]:=TRUE;//出料后,该电芯是MES不良
	END_IF
ELSE
		Alarm_TON[14].IN:=FALSE;
END_IF

IF  CellMemory[CellNo.Thickness].Hough=2 AND Thickness_Finish  AND CellMemory[CellNo.Thickness].Cell AND Step35>=1000 AND Step35<1050  THEN
	IF NOT Alarm_TON[19].Q THEN
		Alarm_TON[19].IN:=TRUE;
	ELSE
			P3_Error[13]:=TRUE;//出料后,该电芯是对齐度不良
	END_IF
ELSE
		Alarm_TON[19].IN:=FALSE;
END_IF

IF  CellMemory[CellNo.Thickness].OvenShift_NG_T  AND Thickness_Finish  AND CellMemory[CellNo.Thickness].Cell AND Step35>=4000 AND Step35<4050  THEN
	IF NOT Alarm_TON[26].Q THEN
		Alarm_TON[26].IN:=TRUE;
	ELSE
			P3_Error[26]:=TRUE;//出料后,该电芯是预热转移时间超时电芯
	END_IF
ELSE
		Alarm_TON[26].IN:=FALSE;
END_IF

IF  CellMemory[CellNo.Thickness].Thickness<>1 AND NOT P3User2_Par.Shield[3] AND Thickness_Finish  AND CellMemory[CellNo.Thickness].Cell AND Step35>=4000 AND Step35<4050  THEN
	IF NOT Alarm_TON[38].Q THEN
		Alarm_TON[38].IN:=TRUE;
	ELSE
			P3_Error[77]:=TRUE;//出料后,该电芯是测厚不良电芯
	END_IF
ELSE
		Alarm_TON[38].IN:=FALSE;
END_IF

IF  CellMemory[CellNo.Thickness].ShortTest<>1 AND NOT P3User2_Par.Shield[1] AND Thickness_Finish  AND CellMemory[CellNo.Thickness].Cell AND Step35>=1000 AND Step35<1050  THEN
	IF NOT Alarm_TON[39].Q THEN
		Alarm_TON[39].IN:=TRUE;
	ELSE
			P3_Error[78]:=TRUE;//出料后,该电芯是短路测试不良
	END_IF
ELSE
		Alarm_TON[39].IN:=FALSE;
END_IF


///////////////////////////////////////////////////////////////////////////////////////////////////////////////////////////////////////////////////////

IF Push_NG_Full[1] THEN
	IF NOT Alarm_TON[15].Q THEN
		Alarm_TON[15].IN:=TRUE;
	ELSE
			P3_Error[9]:=TRUE;//对齐度NG盒满料报警，请人工拿掉料后重新回原
	END_IF
ELSE
		Alarm_TON[15].IN:=FALSE;
END_IF
//报警复位后，判断是否还有料，无料则自动复位
IF P3_Error[9]  AND (P3_SystemRUN.bReset OR stSysState.hmiReset)AND NOT P3Senser.P3_PoleMotor1_bHave THEN
	P3Motion.stP3NgPushMoter[1].bHome:=TRUE;
	P3_Error[9]:=FALSE;
END_IF

IF Push_NG_Full[2] THEN
	IF NOT Alarm_TON[16].Q THEN
		Alarm_TON[16].IN:=TRUE;
	ELSE
			P3_Error[10]:=TRUE;//短路NG盒满料报警，请人工拿掉料后重新回原
	END_IF
ELSE
		Alarm_TON[16].IN:=FALSE;
END_IF
//报警复位后，判断是否还有料，无料则自动复位
IF P3_Error[10]  AND (P3_SystemRUN.bReset OR stSysState.hmiReset)AND NOT P3Senser.P3_PoleMotor2_bHave THEN
	P3Motion.stP3NgPushMoter[2].bHome:=TRUE;
	P3_Error[10]:=FALSE;
END_IF

IF Push_NG_Full[3] THEN
	IF NOT Alarm_TON[17].Q THEN
		Alarm_TON[17].IN:=TRUE;
	ELSE
			P3_Error[11]:=TRUE;//测厚NG盒满料报警，请人工拿掉料后重新回原
	END_IF
ELSE
		Alarm_TON[17].IN:=FALSE;
END_IF
//报警复位后，判断是否还有料，无料则自动复位
IF P3_Error[11]  AND (P3_SystemRUN.bReset OR stSysState.hmiReset)AND NOT P3Senser.P3_PoleMotor3_bHave THEN
	P3Motion.stP3NgPushMoter[3].bHome:=TRUE;
	P3_Error[11]:=FALSE;
END_IF

IF Push_NG_Full[4] THEN
	IF NOT Alarm_TON[18].Q THEN
		Alarm_TON[18].IN:=TRUE;
	ELSE
			P3_Error[12]:=TRUE;//扫码或MES的NG盒满料报警，请人工拿掉料后重新回原
	END_IF
ELSE
		Alarm_TON[18].IN:=FALSE;
END_IF
//报警复位后，判断是否还有料，无料则自动复位
IF P3_Error[12]  AND (P3_SystemRUN.bReset OR stSysState.hmiReset)AND NOT P3Senser.P3_PoleMotor4_bHave THEN
	P3Motion.stP3NgPushMoter[4].bHome:=TRUE;
	P3_Error[12]:=FALSE;
END_IF




IF PC_Error THEN
	P3_Error[14]:=TRUE;//上位机读取PLC数据异常
END_IF

IF (Step35=20 AND CellMemory[CellNo.Weight].Cell AND Permit_Weigh AND NOT Weigh_Finish) AND NOT P3User2_Par.Shield[2] THEN
	IF NOT Alarm_TON[20].Q THEN
		Alarm_TON[20].IN:=TRUE;
	ELSE
		P3_Error[15]:=TRUE;//称重未完成超时报警
		
	END_IF
ELSE
	    Alarm_TON[20].IN:=FALSE;
	
END_IF


//P3_Error[16]已用
//P3_Error[17]已用
//P3_Error[18]已用
//P3_Error[19]已用
 IF NOT  P3Senser.P3_OVenScapegoat1 THEN
	 P3_Error[20]:=TRUE;//烤箱替罪羊1报警
 END_IF

IF NOT  P3Senser.P3_OVenScapegoat2 THEN
	 P3_Error[21]:=TRUE;//烤箱替罪羊2报警
 END_IF
 
 IF NOT  P3Senser.P3_OVenScapegoat3 THEN
	 P3_Error[22]:=TRUE;//烤箱替罪羊3报警
 END_IF

 IF NOT  P3Senser.P3_ColdScapegoat THEN
	 P3_Error[23]:=TRUE;//冷压替罪羊报警
 END_IF
 
 IF NOT  P3Senser.P3_HotScapegoat THEN
	 P3_Error[24]:=TRUE;//热压替罪羊报警
 END_IF
	
 IF arrAxisCtrlV2[P3AxisNo.P3_M2_OvenRetracting].Cmd.arrbRealPoint[43] AND arrAxisCtrlV2[P3AxisNo.P3_M2_OvenRetracting].Status.NoMoving
AND arrAxisCtrlV2[P3AxisNo.P3_M2_OvenRetracting].Status.Homed AND NOT arrAxisCtrlV2[P3AxisNo.P3_M2_OvenRetracting].Io.biHomeSwitch THEN
	 IF NOT Alarm_TON[25].Q THEN
		Alarm_TON[25].IN:=TRUE;
	ELSE
		//P3_Error[25]:=TRUE;//烤箱进退在初始位未感应到原点报警
	END_IF
ELSE
	    Alarm_TON[25].IN:=FALSE;
END_IF
 

 
(*
IF (Step34=105 AND CellMemory[CellNo.WeightClip].Cell AND NOT P3_Weight_gross.Clear_finish) AND NOT P3User2_Par.Shield[2] THEN
	IF NOT Alarm_TON[27].Q THEN
		Alarm_TON[27].IN:=TRUE;
	ELSE
		P3_Error[27]:=TRUE;//称重清零超时报警
		P3_Weight_gross.Init:=TRUE;
	END_IF
ELSE
	    Alarm_TON[27].IN:=FALSE;
	
END_IF
*)
IF Init_step[3]>=1 AND Init_step[3]<=160 AND NOT Oven_CYOFF_condition THEN
	P3_Error[28]:=TRUE;//初始化过程中，烤箱门未完成关闭，请完全关闭再重新启动烤箱初始化
END_IF


//P3_Error[29]已用//冷压条件托板开合不在张开位或者未感应到电芯报警，请复位后确认后再人工启动冷压
//P3_Error[30]已用//热压条件托板开合不在张开位或者未感应到电芯报警，请复位后确认后再人工启动热压
//P3_Error[62]:=P3_Error[29];//冷压空压报警
P3_Error[63]:=P3_Error[30];//热压空压报警

IF  arrCyCtrl[P3CYNo.P3OvenMoveClip].Io.DIOnSwitch THEN//必须把烤箱上料夹感应器，空夹夹紧时的感应器调亮
	IF NOT Alarm_TON[31].Q THEN
		Alarm_TON[31].IN:=TRUE;
	ELSE
		P3_Error[31]:=TRUE;//烤箱上料夹空夹报警
	END_IF
ELSE
	    Alarm_TON[31].IN:=FALSE;
END_IF


IF  arrCyCtrl[P3CYNo.P3WeightFeedingClamp].Io.DIOFFSwitch THEN
	IF NOT Alarm_TON[32].Q THEN
		Alarm_TON[32].IN:=TRUE;
	ELSE
		P3_Error[32]:=TRUE;//称重上料夹空夹报警
	END_IF
ELSE
	    Alarm_TON[32].IN:=FALSE;
END_IF

IF  arrCyCtrl[P3CYNo.P3SortLifting].Io.DIOFFSwitch THEN
	IF NOT Alarm_TON[33].Q THEN
		Alarm_TON[33].IN:=TRUE;
	ELSE
		P3_Error[33]:=TRUE;//分选夹空夹报警
	END_IF
ELSE
	    Alarm_TON[33].IN:=FALSE;
END_IF

IF 	 (stSysState.hmiReset OR P3_SystemRUN.bReset) AND P3_Error[15] THEN
		P3_Weight_gross.Init:=TRUE;
		weight_step:=0;
END_IF



IF arrTempCtrl[1].bSenserError                                        	OR arrTempCtrl[1].bTempError_HI                                  OR
	arrTempCtrl[2].bSenserError                                         OR arrTempCtrl[2].bTempError_HI                                  OR
	arrTempCtrl[3].bSenserError                                         OR arrTempCtrl[3].bTempError_HI                                  OR
	arrTempCtrl[4].bSenserError                                         OR arrTempCtrl[4].bTempError_HI                                  OR
	arrTempCtrl[5].bSenserError                                         OR arrTempCtrl[5].bTempError_HI                                  OR
	arrTempCtrl[6].bSenserError                                         OR arrTempCtrl[6].bTempError_HI                                  OR
	arrTempCtrl[7].bSenserError                                         OR arrTempCtrl[7].bTempError_HI                                  OR
	arrTempCtrl[8].bSenserError                                         OR arrTempCtrl[8].bTempError_HI                                  OR
	arrTempCtrl[9].bSenserError                                         OR arrTempCtrl[9].bTempError_HI                                  OR
	arrTempCtrl[10].bSenserError                                        OR arrTempCtrl[10].bTempError_HI                                 OR
	arrTempCtrl[11].bSenserError                                        OR arrTempCtrl[11].bTempError_HI                                 OR
	arrTempCtrl[12].bSenserError                                        OR arrTempCtrl[12].bTempError_HI                                 OR
	arrTempCtrl[13].bSenserError                                        OR arrTempCtrl[13].bTempError_HI                                 OR
	arrTempCtrl[14].bSenserError                                        OR arrTempCtrl[14].bTempError_HI                                 OR
	arrTempCtrl[15].bSenserError                                        OR arrTempCtrl[15].bTempError_HI                                 OR
	arrTempCtrl[16].bSenserError                                        OR arrTempCtrl[16].bTempError_HI                                 OR
	arrTempCtrl[17].bSenserError                                        OR arrTempCtrl[17].bTempError_HI                                 OR
	arrTempCtrl[18].bSenserError                                        OR arrTempCtrl[18].bTempError_HI                                 OR
	arrTempCtrl[19].bSenserError                                        OR arrTempCtrl[19].bTempError_HI                                 OR
	arrTempCtrl[20].bSenserError                                        OR arrTempCtrl[20].bTempError_HI                                 OR
	arrTempCtrl[21].bSenserError                                        OR arrTempCtrl[21].bTempError_HI                                 OR
	arrTempCtrl[22].bSenserError                                        OR arrTempCtrl[22].bTempError_HI                                 OR
	arrTempCtrl[23].bSenserError                                        OR arrTempCtrl[23].bTempError_HI                                 OR
	arrTempCtrl[24].bSenserError                                        OR arrTempCtrl[24].bTempError_HI                                 OR
	arrTempCtrl[25].bSenserError                                        OR arrTempCtrl[25].bTempError_HI                                 OR
	arrTempCtrl[26].bSenserError                                        OR arrTempCtrl[26].bTempError_HI                                 OR
	arrTempCtrl[27].bSenserError                                        OR arrTempCtrl[27].bTempError_HI                                 OR
	arrTempCtrl[28].bSenserError                                        OR arrTempCtrl[28].bTempError_HI                                 OR
	arrTempCtrl[29].bSenserError                                       (* OR arrTempCtrl[29].bTempError_HI*)                                 OR
	arrTempCtrl[30].bSenserError                                       (* OR arrTempCtrl[30].bTempError_HI*)                                 OR
	arrTempCtrl[31].bSenserError                                        (*OR arrTempCtrl[31].bTempError_HI*)                                 OR
	arrTempCtrl[32].bSenserError                                       (* OR arrTempCtrl[32].bTempError_HI *)                                THEN
		P3Senser.P3_Oven_Power1:=FALSE;
	ELSE
		P3Senser.P3_Oven_Power1:=TRUE;	
	END_IF
	
IF	arrTempCtrl[33].bSenserError                                        OR arrTempCtrl[33].bTempError_HI                                 OR
	arrTempCtrl[34].bSenserError                                        OR arrTempCtrl[34].bTempError_HI                                 OR
	arrTempCtrl[35].bSenserError                                        OR arrTempCtrl[35].bTempError_HI                                 OR
	arrTempCtrl[36].bSenserError                                        OR arrTempCtrl[36].bTempError_HI                                 OR
	arrTempCtrl[37].bSenserError                                        OR arrTempCtrl[37].bTempError_HI                                 OR
	arrTempCtrl[38].bSenserError                                        OR arrTempCtrl[38].bTempError_HI                                 OR
	arrTempCtrl[39].bSenserError                                        OR arrTempCtrl[39].bTempError_HI                                 OR
	arrTempCtrl[40].bSenserError                                        OR arrTempCtrl[40].bTempError_HI                                 OR
	arrTempCtrl[41].bSenserError                                        OR arrTempCtrl[41].bTempError_HI                                 OR
	arrTempCtrl[42].bSenserError                                        OR arrTempCtrl[42].bTempError_HI                                 OR
	arrTempCtrl[43].bSenserError                                        OR arrTempCtrl[43].bTempError_HI                                 OR
	arrTempCtrl[44].bSenserError                                        OR arrTempCtrl[44].bTempError_HI                                 OR
	arrTempCtrl[45].bSenserError                                        OR arrTempCtrl[45].bTempError_HI                                 OR
	arrTempCtrl[46].bSenserError                                        OR arrTempCtrl[46].bTempError_HI                                 OR
	arrTempCtrl[47].bSenserError                                        OR arrTempCtrl[47].bTempError_HI                                 OR
	arrTempCtrl[48].bSenserError                                        OR arrTempCtrl[48].bTempError_HI                                 OR
	arrTempCtrl[49].bSenserError                                        OR arrTempCtrl[49].bTempError_HI                                 OR
	arrTempCtrl[50].bSenserError                                        OR arrTempCtrl[50].bTempError_HI                                 OR
	arrTempCtrl[51].bSenserError                                        OR arrTempCtrl[51].bTempError_HI                                 OR
	arrTempCtrl[52].bSenserError                                        OR arrTempCtrl[52].bTempError_HI                                 OR
	arrTempCtrl[53].bSenserError                                        OR arrTempCtrl[53].bTempError_HI                                 OR
	arrTempCtrl[54].bSenserError                                        OR arrTempCtrl[54].bTempError_HI                                 OR
	arrTempCtrl[55].bSenserError                                        OR arrTempCtrl[55].bTempError_HI                                 OR
	arrTempCtrl[56].bSenserError                                        OR arrTempCtrl[56].bTempError_HI                                 OR
	arrTempCtrl[57].bSenserError                                        OR arrTempCtrl[57].bTempError_HI                                 OR
	arrTempCtrl[58].bSenserError                                        OR arrTempCtrl[58].bTempError_HI                                 OR
	arrTempCtrl[59].bSenserError                                        OR arrTempCtrl[59].bTempError_HI                                 OR
	arrTempCtrl[60].bSenserError                                        OR arrTempCtrl[50].bTempError_HI                                 OR
	arrTempCtrl[61].bSenserError                                        OR arrTempCtrl[51].bTempError_HI                                 OR
	arrTempCtrl[62].bSenserError                                        OR arrTempCtrl[52].bTempError_HI                                 OR
	arrTempCtrl[63].bSenserError                                        OR arrTempCtrl[53].bTempError_HI                                 OR
	arrTempCtrl[64].bSenserError                                        OR arrTempCtrl[54].bTempError_HI                                 OR
	arrTempCtrl[65].bSenserError                                        OR arrTempCtrl[55].bTempError_HI                                 OR
	arrTempCtrl[66].bSenserError                                        OR arrTempCtrl[56].bTempError_HI                                 OR
	arrTempCtrl[67].bSenserError                                        OR arrTempCtrl[57].bTempError_HI                                 OR
	arrTempCtrl[68].bSenserError                                        OR arrTempCtrl[58].bTempError_HI                                 OR
	arrTempCtrl[69].bSenserError                                        OR arrTempCtrl[69].bTempError_HI                                 OR
	arrTempCtrl[70].bSenserError                                        OR arrTempCtrl[70].bTempError_HI                                 OR
	arrTempCtrl[71].bSenserError                                        OR arrTempCtrl[71].bTempError_HI                                 OR
	arrTempCtrl[72].bSenserError                                        OR arrTempCtrl[72].bTempError_HI                                 OR
	arrTempCtrl[73].bSenserError                                        OR arrTempCtrl[73].bTempError_HI                                 OR
	arrTempCtrl[74].bSenserError                                        OR arrTempCtrl[74].bTempError_HI                                 OR
	arrTempCtrl[75].bSenserError                                        OR arrTempCtrl[75].bTempError_HI                                 OR
	arrTempCtrl[76].bSenserError                                        OR arrTempCtrl[76].bTempError_HI                                 OR
	arrTempCtrl[77].bSenserError                                        OR arrTempCtrl[77].bTempError_HI                                 OR
	arrTempCtrl[78].bSenserError                                        OR arrTempCtrl[78].bTempError_HI                                 OR
	arrTempCtrl[79].bSenserError                                        OR arrTempCtrl[79].bTempError_HI                                 OR
	arrTempCtrl[80].bSenserError                                        OR arrTempCtrl[80].bTempError_HI                                 OR
	arrTempCtrl[81].bSenserError                                        OR arrTempCtrl[81].bTempError_HI                                 OR
	arrTempCtrl[82].bSenserError                                        OR arrTempCtrl[82].bTempError_HI                                 OR
	arrTempCtrl[83].bSenserError                                        OR arrTempCtrl[83].bTempError_HI                                 OR
	arrTempCtrl[84].bSenserError                                        OR arrTempCtrl[84].bTempError_HI                                 OR
	arrTempCtrl[85].bSenserError                                        OR arrTempCtrl[85].bTempError_HI                                 OR
	arrTempCtrl[86].bSenserError                                        OR arrTempCtrl[86].bTempError_HI                 				 OR
	arrTempCtrl[87].bSenserError                                        OR arrTempCtrl[87].bTempError_HI                 				 OR
	arrTempCtrl[88].bSenserError                                        OR arrTempCtrl[88].bTempError_HI                 				 OR
	arrTempCtrl[89].bSenserError                                        OR arrTempCtrl[89].bTempError_HI                 				 OR
	arrTempCtrl[90].bSenserError                                        OR arrTempCtrl[90].bTempError_HI                 				 OR
	arrTempCtrl[91].bSenserError                                        OR arrTempCtrl[91].bTempError_HI                 				 OR
	arrTempCtrl[92].bSenserError                                        OR arrTempCtrl[92].bTempError_HI                 				 OR
	arrTempCtrl[93].bSenserError                                        OR arrTempCtrl[93].bTempError_HI                 				 OR
	arrTempCtrl[94].bSenserError                                        OR arrTempCtrl[94].bTempError_HI                 	THEN
		P3Senser.P3_Hotpress_Power:=FALSE;
	ELSE
	 	P3Senser.P3_Hotpress_Power:=TRUE;
	END_IF






//安全门
Door_error[1]:=(NOT P3Senser.P3_Securitydoorswitch1 AND NOT P3User2_Par.Door_Forbidden);
Door_error[2]:=(NOT P3Senser.P3_Securitydoorswitch2 AND NOT P3User2_Par.Door_Forbidden);
Door_error[3]:=(NOT P3Senser.P3_Securitydoorswitch3 AND NOT P3User2_Par.Door_Forbidden);
Door_error[4]:=(NOT P3Senser.P3_Securitydoorswitch4 AND NOT P3User2_Par.Door_Forbidden);
Door_error[5]:=(NOT P3Senser.P3_Securitydoorswitch5 AND NOT P3User2_Par.Door_Forbidden);
Door_error[6]:=(NOT P3Senser.P3_Securitydoorswitch6 AND NOT P3User2_Par.Door_Forbidden);
Door_error[7]:=(NOT P3Senser.P3_Securitydoorswitch7 AND NOT P3User2_Par.Door_Forbidden);
Door_error[8]:=(NOT P3Senser.P3_Securitydoorswitch8 AND NOT P3User2_Par.Door_Forbidden);
Door_error[9]:=(NOT P3Senser.P3_Securitydoorswitch9 AND NOT P3User2_Par.Door_Forbidden);
Door_error[10]:=(NOT P3Senser.P3_Securitydoorswitch10 AND NOT P3User2_Par.Door_Forbidden);
Door_error[11]:=(NOT P3Senser.P3_Securitydoorswitch11 AND NOT P3User2_Par.Door_Forbidden);
Door_error[12]:=(NOT P3Senser.P3_Securitydoorswitch12 AND NOT P3User2_Par.Door_Forbidden);
//Door_error[13]:=(NOT P3Senser.P3_Securitydoorswitch13 AND NOT Door_Forbidden);
//Door_error[14]:=(NOT P3Senser.P3_Securitydoorswitch14 AND NOT Door_Forbidden);
//Door_error[15]:=(NOT P3Senser.P3_Securitydoorswitch15 AND NOT Door_Forbidden);
//Door_error[16]:=(NOT P3Senser.P3_Securitydoorswitch16 AND NOT Door_Forbidden);


//冷压上料平移电机运动过程安全提示
P3Button.P3_ColdWarning_Buzzer:=arrAxisCtrl[P3AxisNo.P3M1_ColdpreLine].Status.Moving;
Twinkle[1].EN:=arrAxisCtrl[P3AxisNo.P3M1_ColdpreLine].Status.Moving;
Twinkle[1].Intervall:=T#200MS;
P3Button.P3_ColdWarning_Lamp:=Twinkle[1].Blink;


//烤箱替罪羊保护
IF NOT  P3Senser.P3_OVenScapegoat1  OR NOT  P3Senser.P3_OVenScapegoat2  OR NOT  P3Senser.P3_OVenScapegoat3 THEN//替罪羊不在轴停止
		arrAxisCtrlV2[P3AxisNo.P3_M2_OvenCarrying].Cmd.bStop:=TRUE;//烤箱搬运轴停止
		arrAxisCtrlV2[P3AxisNo.P3_M2_OvenRetracting].Cmd.bStop:=TRUE;//烤箱进退轴停止
		arrAxisCtrlV2[P3AxisNo.P3_M2_OvenUpDown].Cmd.bStop:=TRUE;//烤箱升降轴停止	
END_IF

IF (stSysState.hmiReset OR P3_SystemRUN.bReset) AND  P3Senser.P3_OVenScapegoat1 AND  P3Senser.P3_OVenScapegoat2 AND  P3Senser.P3_OVenScapegoat3 AND NOT P3_SystemRUN.btnEstop   THEN
		arrAxisCtrlV2[P3AxisNo.P3_M2_OvenCarrying].Cmd.bStop:=FALSE;//烤箱搬运轴停止
		arrAxisCtrlV2[P3AxisNo.P3_M2_OvenRetracting].Cmd.bStop:=FALSE;//烤箱进退轴停止
		arrAxisCtrlV2[P3AxisNo.P3_M2_OvenUpDown].Cmd.bStop:=FALSE;//烤箱升降轴停止	
END_IF


//冷压替罪羊保护
IF NOT P3Senser.P3_ColdScapegoat THEN
	arrAxisCtrl[P3AxisNo.P3M1_ColdpreActuated].Cmd.bStop:=TRUE;
	arrAxisCtrl[P3AxisNo.P3M1_ColdpreSupPlateLine].Cmd.bStop:=TRUE;
END_IF
IF (stSysState.hmiReset OR P3_SystemRUN.bReset) AND P3Senser.P3_ColdScapegoat AND NOT P3_SystemRUN.btnEstop   THEN
		arrAxisCtrl[P3AxisNo.P3M1_ColdpreActuated].Cmd.bStop:=FALSE;
	arrAxisCtrl[P3AxisNo.P3M1_ColdpreSupPlateLine].Cmd.bStop:=FALSE;
END_IF

//热压替罪羊保护
IF NOT P3Senser.P3_HotScapegoat THEN
	arrAxisCtrl[P3AxisNo.P3_M3_HotPressingActuated].Cmd.bStop:=TRUE;
	arrAxisCtrl[P3AxisNo.P3_M3_HotPressingLine].Cmd.bStop:=TRUE;
END_IF
IF (stSysState.hmiReset OR P3_SystemRUN.bReset) AND P3Senser.P3_HotScapegoat AND NOT P3_SystemRUN.btnEstop   THEN
		arrAxisCtrl[P3AxisNo.P3_M3_HotPressingActuated].Cmd.bStop:=FALSE;
		arrAxisCtrl[P3AxisNo.P3_M3_HotPressingLine].Cmd.bStop:=FALSE;
END_IF

//冷压上料轴保护
IF arrAxisCtrl[P3AxisNo.P3M1_ColdpreRetracting].Status.Error OR arrAxisCtrl[P3AxisNo.P3M1_ColdpreLine].Status.Error OR 
	arrAxisCtrl[P3AxisNo.P3M1_ColdpreUpDown].Status.Error OR arrAxisCtrl[P3AxisNo.P3M1_ColdpreWhirling].Status.Error THEN
 		 arrAxisCtrl[P3AxisNo.P3M1_ColdpreRetracting].Cmd.bStop:=TRUE;
		 arrAxisCtrl[P3AxisNo.P3M1_ColdpreLine].Cmd.bStop:=TRUE;
		 arrAxisCtrl[P3AxisNo.P3M1_ColdpreUpDown].Cmd.bStop:=TRUE;
		 arrAxisCtrl[P3AxisNo.P3M1_ColdpreWhirling].Cmd.bStop:=TRUE;		 
END_IF
IF (stSysState.hmiReset OR P3_SystemRUN.bReset) AND  NOT P3_SystemRUN.btnEstop AND
NOT arrAxisCtrl[P3AxisNo.P3M1_ColdpreRetracting].Status.Error AND NOT arrAxisCtrl[P3AxisNo.P3M1_ColdpreLine].Status.Error AND 
NOT arrAxisCtrl[P3AxisNo.P3M1_ColdpreUpDown].Status.Error AND NOT  arrAxisCtrl[P3AxisNo.P3M1_ColdpreWhirling].Status.Error   THEN
		 arrAxisCtrl[P3AxisNo.P3M1_ColdpreRetracting].Cmd.bStop:=FALSE;
		 arrAxisCtrl[P3AxisNo.P3M1_ColdpreLine].Cmd.bStop:=FALSE;
		 arrAxisCtrl[P3AxisNo.P3M1_ColdpreUpDown].Cmd.bStop:=FALSE;
		 arrAxisCtrl[P3AxisNo.P3M1_ColdpreWhirling].Cmd.bStop:=FALSE;		
END_IF

//烤箱轴保护
IF arrAxisCtrlV2[P3AxisNo.P3_M2_OvenCarrying].Status.Error OR arrAxisCtrlV2[P3AxisNo.P3_M2_OvenRetracting].Status.Error OR arrAxisCtrlV2[P3AxisNo.P3_M2_OvenUpDown].Status.Error THEN
	arrAxisCtrlV2[P3AxisNo.P3_M2_OvenCarrying].Cmd.bStop:=TRUE;
	arrAxisCtrlV2[P3AxisNo.P3_M2_OvenRetracting].Cmd.bStop:=TRUE;
	arrAxisCtrlV2[P3AxisNo.P3_M2_OvenUpDown].Cmd.bStop:=TRUE;
END_IF

IF (stSysState.hmiReset OR P3_SystemRUN.bReset) AND  NOT P3_SystemRUN.btnEstop AND
	NOT  arrAxisCtrlV2[P3AxisNo.P3_M2_OvenCarrying].Status.Error AND NOT  arrAxisCtrlV2[P3AxisNo.P3_M2_OvenRetracting].Status.Error 
	AND NOT  arrAxisCtrlV2[P3AxisNo.P3_M2_OvenUpDown].Status.Error THEN
	arrAxisCtrlV2[P3AxisNo.P3_M2_OvenCarrying].Cmd.bStop:=FALSE;
	arrAxisCtrlV2[P3AxisNo.P3_M2_OvenRetracting].Cmd.bStop:=FALSE;
	arrAxisCtrlV2[P3AxisNo.P3_M2_OvenUpDown].Cmd.bStop:=FALSE;
END_IF



//称重上料轴保护
IF arrAxisCtrl[P3AxisNo.P3_M4_WeighLine].Status.Error OR arrAxisCtrl[P3AxisNo.P3_M4_WeighUpDown].Status.Error OR 
	arrAxisCtrl[P3AxisNo.P3_M4_WeighWhirling].Status.Error  THEN
 		 arrAxisCtrl[P3AxisNo.P3_M4_WeighLine].Cmd.bStop:=TRUE;
		 arrAxisCtrl[P3AxisNo.P3_M4_WeighUpDown].Cmd.bStop:=TRUE;
		 arrAxisCtrl[P3AxisNo.P3_M4_WeighWhirling].Cmd.bStop:=TRUE;
END_IF

IF (stSysState.hmiReset OR P3_SystemRUN.bReset) AND  NOT P3_SystemRUN.btnEstop AND
NOT arrAxisCtrl[P3AxisNo.P3_M4_WeighLine].Status.Error AND NOT arrAxisCtrl[P3AxisNo.P3_M4_WeighUpDown].Status.Error AND 
NOT arrAxisCtrl[P3AxisNo.P3_M4_WeighWhirling].Status.Error    THEN
		 arrAxisCtrl[P3AxisNo.P3_M4_WeighLine].Cmd.bStop:=FALSE;
		 arrAxisCtrl[P3AxisNo.P3_M4_WeighUpDown].Cmd.bStop:=FALSE;
		 arrAxisCtrl[P3AxisNo.P3_M4_WeighWhirling].Cmd.bStop:=FALSE;		
END_IF




	
//力矩报警
	IF ColdpreLineTorMark THEN//冷呀上料夹平移力矩超限报警标志
		 IF arrAxisCtrl[P3AxisNo.P3M1_ColdpreLine].Status.Moving AND (ABS(Torque_P3.ColdpreLineTor)>=Torque_P3.ColdpreLineTorSet)  THEN
			HMI_TorAlarm_D[160]:=TRUE;//冷呀上料夹平移力矩超限报警标志
			arrAxisCtrl[P3AxisNo.P3M1_ColdpreLine].Cmd.bEnable:=FALSE;
			//ColdpreLineTorMark:=FALSE;
		END_IF
	END_IF

	IF ColdpreRetractTorMark THEN//冷压上料夹进退力矩超限报警
		 IF arrAxisCtrl[P3AxisNo.P3M1_ColdpreRetracting].Status.Moving AND (ABS(Torque_P3.ColdpreRetractTor)>=Torque_P3.ColdpreRetractTorSet)  THEN
			HMI_TorAlarm_D[161]:=TRUE;//冷压上料夹进退力矩超限报警
			arrAxisCtrl[P3AxisNo.P3M1_ColdpreRetracting].Cmd.bEnable:=FALSE;
			//ColdpreRetractTorMark:=FALSE;
		END_IF
	END_IF
	
	IF ColdpreWhirlTorMark THEN//冷压上料夹旋转力矩超限报警
		 IF arrAxisCtrl[P3AxisNo.P3M1_ColdpreWhirling].Status.Moving AND (ABS(Torque_P3.ColdpreWhirlTor)>=Torque_P3.ColdpreWhirlTorSet)  THEN
			HMI_TorAlarm_D[162]:=TRUE;//冷压上料夹旋转力矩超限报警
			arrAxisCtrl[P3AxisNo.P3M1_ColdpreWhirling].Cmd.bEnable:=FALSE;
			//ColdpreWhirlTorMark:=FALSE;
		END_IF
	END_IF
(*
	IF ColdpreActTorMark THEN//冷压驱动力矩超限报警
		 IF arrAxisCtrl[P3AxisNo.P3M1_ColdpreActuated].Status.Moving AND (ABS(Torque_P3.ColdpreActTor)>=Torque_P3.ColdpreActTorSet)  THEN
			HMI_TorAlarm_D[165]:=TRUE;//冷压驱动力矩超限报警
			arrAxisCtrl[P3AxisNo.P3M1_ColdpreActuated].Cmd.bEnable:=FALSE;
			//ColdpreActTorMark:=FALSE;
		END_IF
	END_IF
*)
	IF OvenCarryTorMark THEN//烤箱上料夹搬运力矩超限报警
		 IF arrAxisCtrl[P3AxisNo.P3_M2_OvenCarrying].Status.Moving AND (ABS(Torque_P3.OvenCarryTor)>=Torque_P3.OvenCarryTorSet)  THEN
			HMI_TorAlarm_D[166]:=TRUE;//烤箱上料夹搬运力矩超限报警
			arrAxisCtrl[P3AxisNo.P3_M2_OvenCarrying].Cmd.bEnable:=FALSE;
			//OvenCarryTorMark:=FALSE;
		END_IF
	END_IF
	
	IF OvenRetractTorMark THEN//烤箱上料夹进退力矩超限报警标志
		 IF arrAxisCtrl[P3AxisNo.P3_M2_OvenRetracting].Status.Moving AND (ABS(Torque_P3.OvenRetractTor)>=Torque_P3.OvenRetractTorSet)  THEN
			HMI_TorAlarm_D[167]:=TRUE;//烤箱上料夹进退力矩超限报警
			arrAxisCtrl[P3AxisNo.P3_M2_OvenRetracting].Cmd.bEnable:=FALSE;
			//OvenRetractTorMark:=FALSE;
		END_IF
	END_IF
(*	
	IF HotpreActTorMark THEN//热压驱动力矩超限报警
		 IF arrAxisCtrl[P3AxisNo.P3_M3_HotPressingActuated].Status.Moving AND (ABS(Torque_P3.HotpreActTor)>=Torque_P3.HotpreActTorSet)  THEN
			HMI_TorAlarm_D[170]:=TRUE;//热压驱动力矩超限报警
			arrAxisCtrl[P3AxisNo.P3_M3_HotPressingActuated].Cmd.bEnable:=FALSE;
			//HotpreActTorMark:=FALSE;
		END_IF
	END_IF
*)
	IF WeighLineTorMark THEN//称重上料夹平移力矩超限报警标志
		 IF arrAxisCtrl[P3AxisNo.P3_M4_WeighLine].Status.Moving AND (ABS(Torque_P3.WeighLineTor)>=Torque_P3.WeighLineTorSet)  THEN
			HMI_TorAlarm_D[171]:=TRUE;//称重上料夹平移力矩超限报警
			arrAxisCtrl[P3AxisNo.P3_M4_WeighLine].Cmd.bEnable:=FALSE;
			//WeighLineTorMark:=FALSE;
		END_IF
	END_IF
	
	IF WeighWhirlTorMark THEN//称重上料夹旋转力矩超限报警标志
		 IF arrAxisCtrl[P3AxisNo.P3_M4_WeighWhirling].Status.Moving AND (ABS(Torque_P3.WeighWhirlTor)>=Torque_P3.WeighWhirlTorSet)  THEN
			HMI_TorAlarm_D[173]:=TRUE;//称重上料夹旋转力矩超限报警
			arrAxisCtrl[P3AxisNo.P3_M4_WeighWhirling].Cmd.bEnable:=FALSE;
			//WeighWhirlTorMark:=FALSE;
		END_IF
	END_IF

	IF SortingCarryTorMark THEN//电芯分选夹搬运力矩超限报警标志
		 IF arrAxisCtrl[P3AxisNo.P3_M4_SortingoutCarrying].Status.Moving AND (ABS(Torque_P3.SortingCarryTor)>=Torque_P3.SortingCarryTorSet)  THEN
			HMI_TorAlarm_D[174]:=TRUE;//电芯分选夹搬运力矩超限报警
			arrAxisCtrl[P3AxisNo.P3_M4_SortingoutCarrying].Cmd.bEnable:=FALSE;
			//SortingCarryTorMark:=FALSE;
		END_IF
	END_IF
	
	IF OffloadCarryTorMark THEN//电芯下料夹搬运报警力矩设定
		 IF arrAxisCtrl[P3AxisNo.P3_M4_OffloadingCarrying].Status.Moving AND (ABS(Torque_P3.OffloadCarryTor)>=Torque_P3.OffloadCarryTorSet)  THEN
			HMI_TorAlarm_D[176]:=TRUE;//电芯下料夹搬运报警力矩报警
			arrAxisCtrl[P3AxisNo.P3_M4_OffloadingCarrying].Cmd.bEnable:=FALSE;
			//OffloadCarryTorMark:=FALSE;
		END_IF
	END_IF

IF NOT arrCyCtrl[P3CYNo.P3TapeVacuo].Io.DIOnSwitch	AND arrCyCtrl[P3CYNo.P3TapeVacuo].Status.ONState  THEN
	IF NOT Alarm_TON[34].Q THEN
		Alarm_TON[34].IN:=TRUE;
	ELSE
		P3_Error[41]	 :=TRUE;//贴胶头真空报警
		arrCyCtrl[P3CYNo.P3TapeVacuo].Cmd.bOFF:=TRUE;//吸胶真空关闭
	END_IF
ELSE
		Alarm_TON[34].IN:=FALSE;
END_IF
(*
IF  P3_SystemRUN.iMode=1  AND  (Step35=605 OR (Step35=520 AND Step38=40))  AND P3Senser.P3_CacheSensor AND arrAxisCtrl[P3AxisNo.P3_M4_SortingoutUpDown].Cmd.arrbRealPoint[1] THEN
	IF NOT Alarm_TON[35].Q  THEN
		Alarm_TON[35].IN:=TRUE;
	ELSE
		P3_Error[43]:=TRUE;//热压后贴胶平台电芯检测传感器检测异常 
	END_IF
ELSE
		Alarm_TON[35].IN:=FALSE;
END_IF
	*)
IF arrCyCtrl[P3CYNo.P3CellSpin].Io.DOStatus1 AND arrCyCtrl[P3CYNo.P3CellPushSpin].Status.OFFState AND NOT arrCyCtrl[P3CYNo.P3CellSpin].Status.ONState THEN
	IF NOT Alarm_TON[36].Q  THEN
		Alarm_TON[36].IN:=TRUE;
	ELSE
		P3_Error[51]:=TRUE;//热压后贴胶旋转气缸180故障报警
	END_IF
ELSE
		Alarm_TON[36].IN:=FALSE;
	
END_IF

IF NOT arrCyCtrl[P3CYNo.P3CellSpin].Io.DOStatus1 AND arrCyCtrl[P3CYNo.P3CellPushSpin].Status.OFFState AND NOT arrCyCtrl[P3CYNo.P3CellSpin].Status.OFFState THEN
	IF NOT Alarm_TON[37].Q  THEN
		Alarm_TON[37].IN:=TRUE;
	ELSE
		P3_Error[52]:=TRUE;//热压后贴胶旋转气缸0故障报警
	END_IF
ELSE
		Alarm_TON[37].IN:=FALSE;
	
END_IF

IF arrCyCtrl[P3CYNo.P3CellPush].Status.Error1                OR arrCyCtrl[P3CYNo.P3CellAdvance].Status.Error1         OR
   arrCyCtrl[P3CYNo.P3TapePush].Status.Error1                OR arrCyCtrl[P3CYNo.P3TapePull].Status.Error1            OR
   arrCyCtrl[P3CYNo.P3TapeLift].Status.Error1                OR arrCyCtrl[P3CYNo.P3TapeCut].Status.Error1             OR
  (* arrCyCtrl[P3CYNo.P3GluePush].Status.Error1              OR*) arrCyCtrl[P3CYNo.P3TapeBuffer].Status.Error1        OR
  arrAxisCtrl[P3AxisNo.P3_TapeAdvance].Status.Error          OR arrAxisCtrl[P3AxisNo.P3_TapeTranslation].Status.Error OR 
   P3_Error[41]                                              OR P3_Error[43]                                          OR
   P3_Error[51]                                              OR P3_Error[52]                                        THEN
   P3_Error[42]	 :=TRUE;//后段贴胶总报警
 END_IF  
 
 
  IF arrAxisCtrl[P3AxisNo.P3_TapeTranslation].Status.Moving AND (ABS(Torque_P3.TapeAdvanceTor)>=Torque_P3.TapeAdvanceTorSet)  THEN
			Torque_P3.TapeAdvanceTorSetAlarm:=TRUE;
			arrAxisCtrl[P3AxisNo.P3_TapeTranslation].Cmd.bEnable:=FALSE;
  END_IF
  
  IF arrAxisCtrl[P3AxisNo.P3_TapeAdvance].Status.Moving AND (ABS(Torque_P3.TapeTranslationTor)>=Torque_P3.TapeTranslationTorSet)  THEN
			Torque_P3.TapeTranslationTorSetAlarm:=TRUE;
			arrAxisCtrl[P3AxisNo.P3_TapeAdvance].Cmd.bEnable:=FALSE;
  END_IF
  
  IF stSysState.hmiReset OR P3_SystemRUN.hmiReset THEN
	  Torque_P3.TapeTranslationTorSetAlarm:=FALSE;
	  Torque_P3.TapeAdvanceTorSetAlarm:=FALSE;
  END_IF
  
//电芯分选夹有料感应器报警
	IF  (Step35=75  OR Step35=585  OR Step35=1050 OR Step35=2050  OR Step35=3060  OR Step35=4100 )  AND NOT P3Senser.P3_Fxjgy AND arrAxisCtrl[P3AxisNo.P3_M4_SortingoutUpDown].Cmd.arrbRealPoint[1] THEN
	   P3_Error[39]:=TRUE;//电芯分选夹未检测到电芯报警
	END_IF

	  
	IF  (Step35=190  OR Step35=515 OR Step35=640 OR Step35=1120 OR Step35=2120 OR Step35=3130 OR Step35=4180 ) AND  P3Senser.P3_Fxjgy AND arrAxisCtrl[P3AxisNo.P3_M4_SortingoutUpDown].Cmd.arrbRealPoint[1] THEN 
		P3_Error[45]:=TRUE;//电芯分选夹检测到电芯报警
	END_IF
	
//冷压上料夹有料感应器报警
IF (Step30=100  OR Step30=1100 OR Step30=2100)AND NOT CellMemory[CellNo.ColdpressClip].Overhang_TF AND NOT P3Senser.P3_Lyslgy THEN
	P3_Error[68]:=TRUE;//冷压上料夹未检测到电芯报警
END_IF
IF (Step30=40 OR Step30=1040 OR Step30=2040 OR Step30=3080 OR Step30=4090)AND  P3Senser.P3_Lyslgy THEN
P3_Error[69]:=TRUE;//冷压上料夹检测到电芯报警
END_IF

//P3_Error[50]热压位电芯位置偏移报警
IF P3_Error[50] AND (P3_SystemRUN.bReset OR stSysState.hmiReset) AND P3_SystemRUN.iMode=3 THEN//
	IF  NOT P3Senser.P3_HotOffset_L THEN
		P3_Error[50]:=FALSE;
	ELSE
		P3_Error[50]:=TRUE;	
	end_if
END_IF
(*
IF P3_Error[50] AND (P3_SystemRUN.bReset OR stSysState.hmiReset)  THEN//寻找Mark孔异常
	IF  NOT P3Senser.P3_HotEmptyPress AND NOT P3Senser.P3_HotOffset_L THEN
		
		MEMSET(ADR(CellMemory[CellNo.Hotpress]),0,SIZEOF(CellMemory[CellNo.Hotpress]));
		Step33:=1;
		Permit_Hot_Press:=FALSE;
		P3_Error[50]:=FALSE;
	ELSE
		P3_Error[50]:=TRUE;	
	end_if
END_IF
*)

IF  CellMemory[CellNo.Weight].Cell  AND NOT P3Senser.P3_WeightSensor AND NOT (Step35>=35 AND Step35<=80)THEN
	P3_Error[53]:=TRUE;//称重台有记忆无电芯报警
END_IF
IF  NOT CellMemory[CellNo.Weight].Cell  AND  P3Senser.P3_WeightSensor AND NOT( Step34>=110 AND Step34<=140) THEN
	P3_Error[54]:=TRUE;//称重台有电芯无记忆报警
END_IF

IF  NOT CellMemory[CellNo.Thickness].Cell  AND  P3Senser.P3_ThicknessSensor AND NOT (Step35>=150 AND Step35<=185) THEN
//	P3_Error[56]:=TRUE;//测厚台有电芯无记忆报警
;
END_IF

IF P3_Error[55] AND  (P3_SystemRUN.bReset OR stSysState.hmiReset) THEN//测厚台有记忆无电芯报警
		P3_Error[55]:=FALSE;
//		Step35:=1;
//		MEMSET(ADR(CellMemory[CellNo.SortClip1]),0,SIZEOF(CellMemory[CellNo.SortClip1]));
END_IF

//Step35=635 记忆传递后检测电芯有无
//Step38=50 放电芯后检测电芯有无
IF P3_SystemRUN.iMode=1 AND CellMemory[CellNo.BlankingPlatform].Cell AND NOT P3Senser.P3_CacheSensor  AND( Step35=635 OR Step38=50) THEN
	 P3_Error[61]:=TRUE;	//后段贴胶有记忆无电芯报警
END_IF
//Step35=605 贴胶放料前检测有无电芯
//Step38=30 流水线取料后检测有无电芯
//Step38=1040 分选轴下降前检测有无电芯
IF P3_SystemRUN.iMode=1 AND P3Senser.P3_CacheSensor AND NOT CellMemory[CellNo.BlankingPlatform].Cell AND (Step38=30 OR Step38=1040 OR (Step35=605 AND  arrAxisCtrl[P3AxisNo.P3_M4_SortingoutUpDown].Cmd.arrbRealPoint[1]))THEN
	  P3_Error[60]:=TRUE;//后段贴胶无记忆有电芯报警
	
END_IF

IF arrCyCtrl[P3CYNo.P3BoxLock1_NG].Status.OFFState   THEN
	tip_6[2]:=TRUE;//电芯NG1料盒锁定气缸未锁定
ELSE
	tip_6[2]:=FALSE;
END_IF
IF arrCyCtrl[P3CYNo.P3BoxLock2_NG].Status.OFFState  THEN
	tip_6[3]:=TRUE;//电芯NG2料盒锁定气缸未锁定
ELSE
	tip_6[3]:=FALSE;
END_IF
IF arrCyCtrl[P3CYNo.P3BoxLock3_NG].Status.OFFState  THEN
	tip_6[4]:=TRUE;//电芯NG3料盒锁定气缸未锁定
ELSE
	tip_6[4]:=FALSE;
END_IF
IF arrCyCtrl[P2CYNo.LockonCy].Status.OFFState  THEN
	tip_6[4]:=TRUE;//电芯对齐度NG料盒锁定气缸未锁定
ELSE
	tip_6[4]:=FALSE;
END_IF
CleanTrig(CLK:= (P3par.CleanTimeHMIHour1 = System.StTime.wHour AND P3par.CleanTimeHMIMin1 =System.stTime.wMinute)
OR	(P3par.CleanTimeHMIHour2 = System.StTime.wHour AND P3par.CleanTimeHMIMin2 =System.stTime.wMinute)
OR	(P3par.CleanTimeHMIHour3 = System.StTime.wHour AND P3par.CleanTimeHMIMin3 =System.stTime.wMinute)
OR	(P3par.CleanTimeHMIHour4 = System.StTime.wHour AND P3par.CleanTimeHMIMin4 =System.stTime.wMinute));

IF	CleanTrig.Q THEN
	P3_Error[59]:=TRUE;//请清洁机台
END_IF

IF NOT P2Senser.P2M1_Coldpressingesensor AND Step30=30 THEN
P3_Error[70]:=TRUE;//冷压上料夹平移到一号叠台贴胶位未到位报警	
END_IF
IF NOT P2Senser.P2M2_Coldpressingesensor AND Step30=1030 THEN
P3_Error[71]:=TRUE;//冷压上料夹平移到二号叠台贴胶位未到位报警	
END_IF
IF NOT P2Senser.P2M3_Coldpressingesensor AND Step30=2030 THEN
P3_Error[72]:=TRUE;//冷压上料夹平移到三号叠台贴胶位未到位报警	
END_IF
IF (P2Senser.P2M1_Coldpressingesensor OR P2Senser.P2M2_Coldpressingesensor OR P2Senser.P2M3_Coldpressingesensor)AND arrAxisCtrl[P3AxisNo.P3M1_ColdpreLine].Cmd.arrbRealPoint[1] THEN
P3_Error[73]:=TRUE;//冷压上料平移一，二，三号叠台处感应器常亮异常报警
END_IF
Alarm_TON[40].IN:=(((NOT CellMemory[CellNo.Gluing1].Overhang_TF AND Step30=60) 
	OR (NOT CellMemory[CellNo.Gluing2].Overhang_TF AND Step30=1060)
	OR (NOT CellMemory[CellNo.Gluing3].Overhang_TF AND Step30=2060))
	AND NOT arrCyCtrl[P3CYNo.P3ColdPressClip].Status.ONState
	AND  arrCyCtrl[P3CYNo.P3ColdPressClip].Status.Error1);
IF Alarm_TON[40].Q THEN
	P3_Error[76]:=TRUE;//冷压上料夹夹正常电芯闭合感应器异常
END_IF



(*  //轴手动对比报警
AxisHandautomatic1(
				Notmoing:=arrAxis[160].Status.NotMoving AND arrAxis[161].Status.NotMoving AND arrAxis[162].Status.NotMoving AND arrAxis[163].Status.NotMoving AND
						  arrAxis[164].Status.NotMoving AND arrAxis[165].Status.NotMoving AND arrAxis[166].Status.NotMoving AND arrAxis[167].Status.NotMoving AND 
						  arrAxis[168].Status.NotMoving AND arrAxis[169].Status.NotMoving AND arrAxis[170].Status.NotMoving AND arrAxis[171].Status.NotMoving AND 
						  arrAxis[172].Status.NotMoving AND arrAxis[173].Status.NotMoving AND arrAxis[174].Status.NotMoving AND arrAxis[175].Status.NotMoving AND 
						  arrAxis[176].Status.NotMoving AND arrAxis[177].Status.NotMoving AND arrAxis[178].Status.NotMoving AND arrAxis[179].Status.NotMoving  AND
                         NOT Coldbusy AND NOT Hotbusy	 , 	
                  Run:= P3_SystemRUN.hmiAuto ,
                  i:=160 , 
                  j:=20,
				  Reset:=LateBlanking_init_start[1] OR  LateBlanking_init_start[2] OR  LateBlanking_init_start[3] OR  LateBlanking_init_start[4] OR  LateBlanking_init_start[5] 
                                 OR  LateBlanking_init_start[6] OR  LateBlanking_init_start[7]  OR  LateBlanking_init_start[8]  , 
                  error=> );
	*)
IF stSysState.hmiReset OR P3_SystemRUN.bReset AND  NOT (P3_Error[107] OR P3_Error[101] OR P3_Error[102] ) THEN
	b_Alarm[4]:=FALSE;
	PC_Error:=FALSE;
	bCodeConError:=FALSE;
	bCodeError:=FALSE;
	MEMSET(ADR(P3_Error),0,SIZEOF(P3_Error));
	MEMSET(ADR(tip_10),0,SIZEOF(tip_10));
	MEMSET(ADR(Door_error),0,SIZEOF(Door_error)); 
	MEMSET(ADR(P3_Tem_Error),0,SIZEOF(P3_Tem_Error)); 
END_IF

ACTION Alarm:
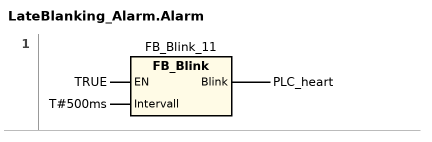
// NETWORK 1
FB_Blink_11(EN := TRUE, Intervall := T#500ms); // FB_Blink
PLC_heart := FB_Blink_11.Blink;
END_ACTION

END_PROGRAM

// ---- P3POUs/P3FB/FB_Blink.TcPOU
FUNCTION_BLOCK FB_Blink   //脉冲发生器
VAR_INPUT
	EN:			BOOL;
	Intervall:		TIME;
END_VAR
VAR_OUTPUT
	Blink:		BOOL;
END_VAR
VAR
	TON_01:		TON;
	TON_02:		TON;
END_VAR

IF EN THEN
	TON_01	(IN:=	NOT TON_02.Q, PT:=Intervall);
	TON_02	(IN:=	 TON_01.Q, PT:=Intervall);
	Blink:= TON_01.Q;
ELSE
	Blink := FALSE;
END_IF

END_FUNCTION_BLOCK

// ---- P3POUs/P3FB/FB_AxisHandautomatic_1.TcPOU
FUNCTION_BLOCK FB_AxisHandautomatic_1
VAR_INPUT
    Notmoing:BOOL;//主轴停止中
	Run:BOOL;//自动
	i:INT;
	j: INT;
	Reset:BOOL;//手自动对比复位
END_VAR

VAR_OUTPUT
error :BOOL ;
END_VAR

VAR
	step:INT ;
	rRun : R_TRIG;
	fRun: F_TRIG;

	Pause_CMD:ARRAY[1..185] OF LREAL ; //手自动对比位置
	Handautomark:BOOL;//手自动对比标志
	K: INT;
	K1: INT;

END_VAR

VAR_IN_OUT

END_VAR




rRun(CLK:= Run , Q=> );
fRun(CLK:= Run , Q=> );


		IF fRun.Q THEN
			step:=100; 
		END_IF
		
	CASE step OF	
		100:
		   IF Notmoing THEN
			 step:=110;  
		   END_IF
	    110:    
	        Handautomark:=TRUE;
			FOR K:=i TO ((i+j)-1) DO 
				IF   K<>166 AND K<>167 AND K<>168  THEN
			          Pause_CMD[K]:=arrAxisCtrl[K].Status.fActPos;
				END_IF	  
			END_FOR
			Pause_CMD[166]:=arrAxisCtrlV2[166].Status.fActPos;
			Pause_CMD[167]:=arrAxisCtrlV2[167].Status.fActPos;
			Pause_CMD[168]:=arrAxisCtrlV2[168].Status.fActPos;
			
	        step:=120;    
	END_CASE
		

	   IF rRun.Q AND Handautomark THEN
				FOR K:=i TO ((i+j)-1) DO 
						IF  ABS(Pause_CMD[K]-arrAxisCtrl[K].Status.fActPos)>=0.2 AND K<>166 AND K<>167 AND K<>168  THEN
						Axis_error[k]:=TRUE;
						END_IF
			
						IF  ABS(Pause_CMD[166]-arrAxisCtrlV2[166].Status.fActPos)>0.2  THEN
						Axis_error[166]:=TRUE;
						END_IF

						IF  ABS(Pause_CMD[167]-arrAxisCtrlV2[167].Status.fActPos)>0.2  THEN
						Axis_error[167]:=TRUE;
						END_IF

						IF  ABS(Pause_CMD[168]-arrAxisCtrlV2[168].Status.fActPos)>0.2  THEN
						Axis_error[168]:=TRUE;
						END_IF
			
						IF Axis_error[k]   THEN
							error:=TRUE;
						END_IF
				END_FOR
				    Handautomark:=FALSE;
		END_IF
		
		IF stSysState.btnReset OR  stSysState.hmiReset  THEN
			   error:=FALSE;
			   FOR K1:=1 TO 185 DO 
				       Axis_error [K1]:=FALSE;
			   END_FOR
		END_IF
		
		IF Reset THEN
			 Handautomark:=FALSE;
		END_IF

END_FUNCTION_BLOCK

// ---- P3POUs/P3FB/ShortTest.TcPOU
FUNCTION_BLOCK ShortTest
VAR_INPUT
	//ShortCircuit---短路
END_VAR
VAR_IN_OUT
	TestCtrl:ShortTestCtrl;//测试控制
	T_Send :ST_SendTestStatus;//发送状态控制字
	T_Receive:ST_ReceiveTestStatus;//接收状态控制字
	
	uSendData:ShortTestSendData;//发送数据命令(STRING转ASCLL)
	uReceiveData:ShortTestReceiveData;//接收数据(ASCLL转string)
	
END_VAR

VAR_OUTPUT
	
	DataError1:BOOL;//电阻值返回数据异常
	DataError2:BOOL;//电压值返回数据异常
	DataError3:BOOL;//测试时间返回数据异常
	DataError4:BOOL;//初始化异常
END_VAR
VAR
	L_R:UDINT;//返回数据的长度
	AutoStep:UINT;//主程序步
	InitStep:UINT;//初始化步
	Test_TON :ARRAY[1..6] OF TON;//延时
	
	
(*发送*)
	sTestSendCmd	:STRING;//命令1字发送字符串
	sTestSend1Cmd	:STRING;//命令1字符串,电阻值：MEASure
	sTestSend2Cmd	:STRING;//命令2字符串,电压值:VOLTage
	sTestSend3Cmd	:STRING;//命令3字符串,短路结果:SHORtcheck:RESult？
(*接收*)
	sCmdReceive		:STRING;//命令返回数据
	sCmd1Receive	:REAL;//命令1返回数据,电阻值
	sCmd2Receive	:REAL;//命令2返回数据,电压值
	sCmd3Receive	:REAL;//命令3返回数据,短路结果
	
//>=32位数据长度,<=64字节	
	SendData1:STRING;//数据长度大于32，小于64，第一次需要发送的数据
	SendData2:STRING;//数据长度大于32，小于64，第二次需要发送的数据
	ReceiveData1:STRING;(*第一次接收到的数据*)
	ReceiveData2:STRING;(*第二次接收到的数据*)
	
	
	L_sCmdReceive1:INT;//电阻值数据长度
	L_sCmdReceive2:INT;//电压值数据长度
	
	sCmdReceive1_DEL:STRING;//第二三个返回数据截取缓存
	sCmdReceive2_DEL:STRING;//第3个数据截取缓存
	
	TestTON:ARRAY[1..3] OF TON;
	

	aaaa: BOOL;
END_VAR





ACT01_Test();
IF P3_SystemRUN.iMode=3THEN
	ACT02_Init();
END_IF

ACTION ACT01_Test:
//命令添加，注意顺序
	sTestSend1Cmd	:=':MEASure?$R;';//命令1字符串,电阻值：MEASure
	sTestSend2Cmd	:=':VOLTage?$R;';//命令2字符串,电压值:VOLTage
	//sTestSend3Cmd	:=':TIMer?$R;';//命令3字符串,测试时间
	//sTestSend3Cmd	:=':DELay?$R;';//命令3字符串,测试时间
	//uSendData.sData :=concat(sTestSend1Cmd,concat());
	sTestSend3Cmd	:=':TIMer?$R;';//命令3字符串,测试时间
CASE AutoStep  OF	
0:
	uSendData.sData:=':MOHM:AUTO:DCLear OFF';
	T_Send.OutputLength:=INT_TO_UINT (LEN(uSendData.sData));//发送数据长度
	AutoStep:=20;
20:
	T_Send.TransmitRequest:=TRUE;
	T_Send.PutData:=TRUE;	
	AutoStep:=50;	
50:
	IF  T_Receive.TransmitDone THEN//数据发送完成
		AutoStep:=80;
	END_IF
80:
	T_Send.PutData:=FALSE;	
	T_Send.TransmitRequest:=FALSE;
	IF NOT T_Send.PutData THEN
		AutoStep:=100;
	END_IF
100://	串口初始化
	T_Send.InitRequest:=TRUE;//
	IF T_Receive.InitAccepted THEN
		T_Send.InitRequest:=FALSE;//
		AutoStep:=200;
	END_IF
200://发送，结束数据缓存区初始化
	sTestSendCmd:='';//命令1字发送字符串
	sCmdReceive:='';//命令返回数据
	sCmd1Receive:=0;
	sCmd2Receive:=0;
	sCmd3Receive:=0;
	uSendData.sData :='';
	uReceiveData.sData:='';
	TestCtrl.bDone:=FALSE;
	MEMSET(ADR(uSendData),0,SIZEOF(uSendData));
	AutoStep:=300;
300:
	IF TestCtrl.bStart THEN
		AutoStep:=400;	
	END_IF
400:
	
	TestCtrl.bDone :=FALSE;	//读取完成
	AutoStep:=500;	
500:
	uSendData.sData:=sTestSend1Cmd;//发送数据
	T_Send.OutputLength:=INT_TO_UINT (LEN(uSendData.sData));//发送数据长度
	AutoStep:=600;	
600:
	T_Send.TransmitRequest:=TRUE;
	T_Send.PutData:=TRUE;	
	AutoStep:=700;	
700:
	IF  T_Receive.TransmitDone THEN//数据发送完成
		AutoStep:=800;
	END_IF
800:
	Test_TON[1](IN:=FALSE);
	T_Send.PutData:=FALSE;	
	T_Send.TransmitRequest:=FALSE;
	IF NOT T_Send.PutData THEN
		AutoStep:=900;	//等待数据返回 
	END_IF
	
900://等待数据	
	Test_TON[1](IN:=TRUE , PT:=T#1.5S , Q=> , ET=> );
	IF T_Receive.ReceiveRequest   THEN//可以接收数据
		AutoStep:=950;	//等待数据返回 
	ELSIF Test_TON[1].Q THEN
		Test_TON[1](IN:=FALSE);
		AutoStep:=100;
	END_IF
950:
	IF T_Receive.TotalInputLength>=2 THEN
		AutoStep:=1000;	//等待数据返回 
	ELSE
		DataError1:=TRUE;//电阻值反悔哦数据异常
	END_IF	
1000:
	T_Send.ReceiveAccepted:=TRUE;//请求读取
	AutoStep:=1100;	//等待数据返回 	
1100://判断数据长度
	IF T_Receive.TotalInputLength<=32 THEN
		AutoStep:=1200;	//等待数据返回 	
	END_IF
1200:
	sCmd1Receive:=STRING_TO_REAL(uReceiveData.sData);//命令返回数据
	AutoStep:=1300;	//等待数据返回 	
1300:
	T_Send.ReceiveAccepted:=TRUE;
	IF NOT T_Receive.ReceiveRequest THEN
		T_Send.ReceiveAccepted:=FALSE;	
		AutoStep:=1400;
	END_IF
1400:
	T_Send.InitRequest:=TRUE;//
	IF T_Receive.InitAccepted THEN
		T_Send.InitRequest:=FALSE;//
		AutoStep:=2000;
	END_IF

2000:
	uSendData.sData:=sTestSend2Cmd;//发送数据
	T_Send.OutputLength:=INT_TO_UINT (LEN(uSendData.sData));//发送数据长度
	AutoStep:=2100;	
2100:
	T_Send.TransmitRequest:=TRUE;
	T_Send.PutData:=TRUE;	
	AutoStep:=2200;	
2200:
	IF  T_Receive.TransmitDone THEN//数据发送完成
		AutoStep:=2300;
	END_IF
2300:
	T_Send.PutData:=FALSE;	
	T_Send.TransmitRequest:=FALSE;
	IF NOT T_Send.PutData THEN
		AutoStep:=2400;	//等待数据返回 
	END_IF
	
2400://等待数据	
	IF T_Receive.ReceiveRequest  THEN//可以接收数据
		AutoStep:=2450;	//等待数据返回 
	END_IF
2450:
	IF  T_Receive.TotalInputLength>=2 THEN
		AutoStep:=2500;	//等待数据返回 
	ELSE
		DataError2:=TRUE;//电压值返回数据异常
	END_IF
2500:
	T_Send.ReceiveAccepted:=TRUE;//请求读取
	AutoStep:=2600;	//等待数据返回 	
2600://判断数据长度
	IF T_Receive.TotalInputLength<=32 THEN
		AutoStep:=2700;	//等待数据返回 	
	END_IF
2700:
	sCmd2Receive:=STRING_TO_REAL(uReceiveData.sData);//命令返回数据
	AutoStep:=2800;	//等待数据返回 	
2800:
	T_Send.ReceiveAccepted:=TRUE;
	IF NOT T_Receive.ReceiveRequest THEN
		T_Send.ReceiveAccepted:=FALSE;	
		AutoStep:=2900;
	END_IF
2900:
	T_Send.InitRequest:=TRUE;//
	IF T_Receive.InitAccepted THEN
		T_Send.InitRequest:=FALSE;//
		AutoStep:=3000;
	END_IF
3000:
	uSendData.sData:=sTestSend3Cmd;//发送数据
	T_Send.OutputLength:=INT_TO_UINT (LEN(uSendData.sData)+1);//发送数据长度
	AutoStep:=3100;	
3100:
	T_Send.TransmitRequest:=TRUE;
	T_Send.PutData:=TRUE;	
	AutoStep:=3200;	
3200:
	IF  T_Receive.TransmitDone THEN//数据发送完成
		AutoStep:=3300;
	END_IF
3300:
	T_Send.PutData:=FALSE;	
	T_Send.TransmitRequest:=FALSE;
	IF NOT T_Send.PutData THEN
		AutoStep:=3400;	//等待数据返回 
	END_IF
	
3400://等待数据	
	IF T_Receive.ReceiveRequest  THEN//可以接收数据
		AutoStep:=3450;	//等待数据返回 
	END_IF
3450:
	IF  T_Receive.TotalInputLength>=2 THEN
		AutoStep:=3500;	//等待数据返回 
	ELSE
		DataError3:=TRUE;//测试时间返回异常
	END_IF
3500:
	T_Send.ReceiveAccepted:=TRUE;//请求读取
	AutoStep:=3600;	//等待数据返回 	
3600://判断数据长度
	IF T_Receive.TotalInputLength<=32 THEN
		AutoStep:=3700;	//等待数据返回 	
	END_IF
3700:
	sCmd3Receive:=STRING_TO_REAL(uReceiveData.sData);//命令返回数据
	AutoStep:=3800;	//等待数据返回 	
	
3800:
	T_Send.ReceiveAccepted:=TRUE;
	IF NOT T_Receive.ReceiveRequest  THEN
		T_Send.ReceiveAccepted:=FALSE;	
		AutoStep:=3900;
	END_IF
3900:
	T_Send.InitRequest:=TRUE;//
	IF T_Receive.InitAccepted THEN
		T_Send.InitRequest:=FALSE;//
		AutoStep:=5000;
	END_IF
5000:
	TestCtrl.Measure:=sCmd1Receive;//电阻值
	TestCtrl.Voltage:=sCmd2Receive;//电压值
	TestCtrl.TestTime:=sCmd3Receive;//测试时间//sCmd3Receive
	AutoStep:=5100;





5100://数据读取完成，允许数据绑定
	TestCtrl.bStart :=FALSE;//读取开始
	TestCtrl.bDone:=TRUE;//数据上传完成
	AutoStep:=6000;
6000:
	IF NOT TestCtrl.bDone THEN
		AutoStep:=100;
	END_IF 
END_CASE






	
(*	
600://发送数据转换为ASCLL码
	IF  T_Send.OutputLength<=32 THEN//数据长度小于32字节
		AutoStep:=700;	
	ELSE
		AutoStep:=1000;
	END_IF	
700:
	//uSendData.sData:=sTestSendCmd;//发送数据
	AutoStep:=800;	
800:
	T_Send.TransmitRequest:=TRUE;
	T_Send.PutData:=TRUE;	
	AutoStep:=900;	
900:
	IF  T_Receive.TransmitDone THEN//数据发送完成
		AutoStep:=950;
	END_IF
950:
	T_Send.PutData:=FALSE;	
	T_Send.TransmitRequest:=FALSE;
	IF NOT T_Send.PutData THEN
		AutoStep:=3000;	//等待数据返回 
	END_IF

1000://数据长度大于32
	T_Send.OutputLength:=INT_TO_UINT (LEN(uSendData.sData));//发送数据长度,32<=L<=64
	SendData1:=LEFT(uSendData.sData,32);//数据长度大于32，小于64，第一次需要发送的数据
	SendData2:=DELETE(uSendData.sData,32,1);//数据长度大于32，小于64，第二次需要发送的数据
	AutoStep:=1100;
1100://第一次数据发送
	uSendData.sData:=SendData1;//发送数据
	AutoStep:=1200;		
1200:
	T_Send.TransmitRequest:=TRUE;
	T_Send.PutData:=TRUE;	
	AutoStep:=1300;		
1300:
	IF  T_Receive.PutDataDone THEN
		T_Send.PutData:=FALSE;	
		AutoStep:=1400;
	END_IF
1400://第二次发送
	uSendData.sData:=SendData2;//发送数据
	AutoStep:=1500;
1500:
	T_Send.PutData:=TRUE;	
	AutoStep:=1600;
1600:
	IF  T_Receive.TransmitDone THEN//数据发送完成
		AutoStep:=1700;
	END_IF
	
1700:
	T_Send.PutData:=FALSE;	
	T_Send.TransmitRequest:=FALSE;
	IF NOT T_Send.PutData THEN
		AutoStep:=3000;	//等待数据返回 
	END_IF 

3000://等待数据	
	IF T_Receive.ReceiveRequest AND T_Receive.TotalInputLength>=6 THEN//可以接收数据
		AutoStep:=3100;	//等待数据返回 
	ELSE
		DataError1:=TRUE;//数据1异常报警
	END_IF
3100:
	T_Send.ReceiveAccepted:=TRUE;//请求读取
	AutoStep:=3150;	//等待数据返回 	
3150://判断数据长度
	IF T_Receive.TotalInputLength<=32 THEN
		AutoStep:=3200;	//等待数据返回 	
	ELSE//数据长度>=32
		AutoStep:=3500;	//等待数据返回 
	END_IF
3200:
	sCmdReceive:=uReceiveData.sData;//命令返回数据
	AutoStep:=3300;	//等待数据返回 	
3300:
	T_Send.ReceiveAccepted:=TRUE;
	IF NOT T_Receive.ReceiveRequest THEN
		T_Send.ReceiveAccepted:=FALSE;	
		AutoStep:=5000;	//等待数据返回 	
	END_IF
	

3500:
	ReceiveData1:=uReceiveData.sData;(*第一次接收到的数据*)
	AutoStep:=3600;	//等待数据返回
3600:
	T_Send.ReceiveAccepted:=TRUE;
	IF NOT T_Receive.ReceiveRequest THEN  	
		T_Send.ReceiveAccepted:=FALSE;	
		AutoStep:=3700;	//等待数据返回
	END_IF
3700:
	IF T_Receive.ReceiveRequest THEN
		ReceiveData2:=uReceiveData.sData;(*第二次接收到的数据*)
		AutoStep:=3800;	//等待数据返回
	END_IF
3800:
	T_Send.ReceiveAccepted:=TRUE;
	IF NOT T_Receive.ReceiveRequest THEN
		T_Send.ReceiveAccepted:=FALSE;	
		AutoStep:=3900;	//等待数据返回 	
	END_IF
3900:
	sCmdReceive:=CONCAT(ReceiveData1,ReceiveData2);//命令返回数据
	AutoStep:=5000;	//等待数据返回 	
	

5000://返回数据开始解码
//电阻值
	L_sCmdReceive1:=FIND(sCmdReceive,';');//电阻值数据长度
	sCmd1Receive:=LEFT(sCmdReceive,L_sCmdReceive1);//电阻值数据
//电压值，短路测试结果
	sCmdReceive1_DEL:=DELETE(sCmdReceive,(L_sCmdReceive1),1);
	L_sCmdReceive2:=FIND(sCmdReceive1_DEL,';');//电压值数据长度
	sCmd2Receive:=LEFT(sCmdReceive1_DEL,L_sCmdReceive2);//命令2返回数据,电压值
//短路测试结果截取	
	sCmdReceive2_DEL:=DELETE(sCmdReceive1_DEL,(L_sCmdReceive2),1);//第3个数据截取缓存
	sCmd3Receive:=sCmdReceive2_DEL;//命令3返回数据,测试时间
	AutoStep:=5100;
*)
END_ACTION

ACTION ACT02_Init:
CASE InitStep OF//初始化步

0:
	InitStep:=100;
100:
	IF TestCtrl.Init  THEN
		TestCtrl.InitFinish:=FALSE;//初始化完成
		InitStep:=105;
	END_IF
105:
	IF NOT TestCtrl.InitFinish THEN
		InitStep:=110;	
	END_IF
110:
	T_Send.InitRequest:=TRUE;//
	IF T_Receive.InitAccepted THEN
		T_Send.InitRequest:=FALSE;//
		InitStep:=200;
	END_IF
200:	
	TestCtrl.Init:=FALSE;
	//TestCtrl.bStart:=FALSE;
	TestCtrl.bDone:=FALSE;
	uSendData.sData:='';
	uReceiveData.sData :='';
	InitStep:=300;
300://仪器初始化
	uSendData.sData:='*RST$R';
	T_Send.OutputLength:=INT_TO_UINT (LEN(uSendData.sData));//发送数据长度
	InitStep:=400;
400:
	T_Send.TransmitRequest:=TRUE;
	T_Send.PutData:=TRUE;	
	InitStep:=500;	
500:
	TestTON[3](IN:=TRUE,PT:=T#2S);
	IF  T_Receive.TransmitDone THEN//数据发送完成
		TestTON[3](IN:=FALSE);
		DataError4:=FALSE;//测试仪初始化异常
		InitStep:=600;
	ELSIF TestTON[3].Q THEN
		TestTON[3].IN :=FALSE;
		DataError4:=TRUE;//测试仪初始化异常
	END_IF
600:
	DataError1:=FALSE;
	DataError2:=FALSE;
	DataError3:=FALSE;
	T_Send.PutData:=FALSE;	
	T_Send.TransmitRequest:=FALSE;
	IF NOT T_Send.PutData THEN
		InitStep:=700;	//等待数据返回 
	END_IF
	
700:
	AutoStep:=0;	
	TestCtrl.InitFinish:=TRUE;//初始化完成
	InitStep:=2000;	//等待数据返回 
2000:
	InitStep:=0;
	
	
END_CASE
END_ACTION

END_FUNCTION_BLOCK

// ---- P3POUs/POUs/Auxiliary/LateBlanking_Condition.TcPOU
PROGRAM LateBlanking_Condition
VAR
	aaa :BOOL;
END_VAR


//烤箱电芯记忆 
IF CellMemory[CellNo.Oven_M1].Cell THEN
	P3User2_Par.Oven_cell[1]:=TRUE;
	ELSE
	P3User2_Par.Oven_cell[1]:=FALSE;	
END_IF
IF CellMemory[CellNo.Oven_M2].Cell THEN
	P3User2_Par.Oven_cell[2]:=TRUE;
	ELSE
	P3User2_Par.Oven_cell[2]:=FALSE;	
END_IF
IF CellMemory[CellNo.Oven_M3].Cell THEN
	P3User2_Par.Oven_cell[3]:=TRUE;
	ELSE
	P3User2_Par.Oven_cell[3]:=FALSE;	
END_IF
IF CellMemory[CellNo.Oven_M4].Cell THEN
	P3User2_Par.Oven_cell[4]:=TRUE;
	ELSE
	P3User2_Par.Oven_cell[4]:=FALSE;	
END_IF
IF CellMemory[CellNo.Oven_M5].Cell THEN
	P3User2_Par.Oven_cell[5]:=TRUE;
	ELSE
	P3User2_Par.Oven_cell[5]:=FALSE;	
END_IF
IF CellMemory[CellNo.Oven_M6].Cell THEN
	P3User2_Par.Oven_cell[6]:=TRUE;
	ELSE
	P3User2_Par.Oven_cell[6]:=FALSE;	
END_IF
IF CellMemory[CellNo.Oven_M7].Cell THEN
	P3User2_Par.Oven_cell[7]:=TRUE;
	ELSE
	P3User2_Par.Oven_cell[7]:=FALSE;	
END_IF
IF CellMemory[CellNo.Oven_M8].Cell THEN
	P3User2_Par.Oven_cell[8]:=TRUE;
	ELSE
	P3User2_Par.Oven_cell[8]:=FALSE;	
END_IF
IF CellMemory[CellNo.Oven_M9].Cell THEN
	P3User2_Par.Oven_cell[9]:=TRUE;
	ELSE
	P3User2_Par.Oven_cell[9]:=FALSE;	
END_IF
IF CellMemory[CellNo.Oven_M10].Cell THEN
	P3User2_Par.Oven_cell[10]:=TRUE;
	ELSE
	P3User2_Par.Oven_cell[10]:=FALSE;	
END_IF
IF CellMemory[CellNo.Oven_M11].Cell THEN
	P3User2_Par.Oven_cell[11]:=TRUE;
	ELSE
	P3User2_Par.Oven_cell[11]:=FALSE;	
END_IF
IF CellMemory[CellNo.Oven_M12].Cell THEN
	P3User2_Par.Oven_cell[12]:=TRUE;
	ELSE
	P3User2_Par.Oven_cell[12]:=FALSE;	
END_IF
IF CellMemory[CellNo.Oven_M13].Cell THEN
	P3User2_Par.Oven_cell[13]:=TRUE;
	ELSE
	P3User2_Par.Oven_cell[13]:=FALSE;	
END_IF
IF CellMemory[CellNo.Oven_M14].Cell THEN
	P3User2_Par.Oven_cell[14]:=TRUE;
	ELSE
	P3User2_Par.Oven_cell[14]:=FALSE;	
END_IF
IF CellMemory[CellNo.Oven_M15].Cell THEN
	P3User2_Par.Oven_cell[15]:=TRUE;
	ELSE
	P3User2_Par.Oven_cell[15]:=FALSE;	
END_IF
IF CellMemory[CellNo.Oven_M16].Cell THEN
	P3User2_Par.Oven_cell[16]:=TRUE;
	ELSE
	P3User2_Par.Oven_cell[16]:=FALSE;	
END_IF
IF CellMemory[CellNo.Oven_M17].Cell THEN
	P3User2_Par.Oven_cell[17]:=TRUE;
	ELSE
	P3User2_Par.Oven_cell[17]:=FALSE;	
END_IF
IF CellMemory[CellNo.Oven_M18].Cell THEN
	P3User2_Par.Oven_cell[18]:=TRUE;
	ELSE
	P3User2_Par.Oven_cell[18]:=FALSE;	
END_IF
IF CellMemory[CellNo.Oven_M19].Cell THEN
	P3User2_Par.Oven_cell[19]:=TRUE;
	ELSE
	P3User2_Par.Oven_cell[19]:=FALSE;	
END_IF
IF CellMemory[CellNo.Oven_M20].Cell THEN
	P3User2_Par.Oven_cell[20]:=TRUE;
	ELSE
	P3User2_Par.Oven_cell[20]:=FALSE;	
END_IF
IF CellMemory[CellNo.Oven_M21].Cell THEN
	P3User2_Par.Oven_cell[21]:=TRUE;
	ELSE
	P3User2_Par.Oven_cell[21]:=FALSE;	
END_IF
IF CellMemory[CellNo.Oven_M22].Cell THEN
	P3User2_Par.Oven_cell[22]:=TRUE;
	ELSE
	P3User2_Par.Oven_cell[22]:=FALSE;	
END_IF
IF CellMemory[CellNo.Oven_M23].Cell THEN
	P3User2_Par.Oven_cell[23]:=TRUE;
	ELSE
	P3User2_Par.Oven_cell[23]:=FALSE;	
END_IF
IF CellMemory[CellNo.Oven_M24].Cell THEN
	P3User2_Par.Oven_cell[24]:=TRUE;
	ELSE
	P3User2_Par.Oven_cell[24]:=FALSE;	
END_IF
IF CellMemory[CellNo.Oven_M25].Cell THEN
	P3User2_Par.Oven_cell[25]:=TRUE;
	ELSE
	P3User2_Par.Oven_cell[25]:=FALSE;	
END_IF
IF CellMemory[CellNo.Oven_M26].Cell THEN
	P3User2_Par.Oven_cell[26]:=TRUE;
	ELSE
	P3User2_Par.Oven_cell[26]:=FALSE;	
END_IF
IF CellMemory[CellNo.Oven_M27].Cell THEN
	P3User2_Par.Oven_cell[27]:=TRUE;
	ELSE
	P3User2_Par.Oven_cell[27]:=FALSE;	
END_IF
IF CellMemory[CellNo.Oven_M28].Cell THEN
	P3User2_Par.Oven_cell[28]:=TRUE;
	ELSE
	P3User2_Par.Oven_cell[28]:=FALSE;	
END_IF
IF CellMemory[CellNo.Oven_M29].Cell THEN
	P3User2_Par.Oven_cell[29]:=TRUE;
	ELSE
	P3User2_Par.Oven_cell[29]:=FALSE;	
END_IF
IF CellMemory[CellNo.Oven_M30].Cell THEN
	P3User2_Par.Oven_cell[30]:=TRUE;
	ELSE
	P3User2_Par.Oven_cell[30]:=FALSE;	
END_IF
IF CellMemory[CellNo.Oven_M31].Cell THEN
	P3User2_Par.Oven_cell[31]:=TRUE;
	ELSE
	P3User2_Par.Oven_cell[31]:=FALSE;	
END_IF
IF CellMemory[CellNo.Oven_M32].Cell THEN
	P3User2_Par.Oven_cell[32]:=TRUE;
	ELSE
	P3User2_Par.Oven_cell[32]:=FALSE;	
END_IF
IF CellMemory[CellNo.Oven_M33].Cell THEN
	P3User2_Par.Oven_cell[33]:=TRUE;
	ELSE
	P3User2_Par.Oven_cell[33]:=FALSE;	
END_IF
IF CellMemory[CellNo.Oven_M34].Cell THEN
	P3User2_Par.Oven_cell[34]:=TRUE;
	ELSE
	P3User2_Par.Oven_cell[34]:=FALSE;	
END_IF
IF CellMemory[CellNo.Oven_M35].Cell THEN
	P3User2_Par.Oven_cell[35]:=TRUE;
	ELSE
	P3User2_Par.Oven_cell[35]:=FALSE;	
END_IF
IF CellMemory[CellNo.Oven_M36].Cell THEN
	P3User2_Par.Oven_cell[36]:=TRUE;
	ELSE
	P3User2_Par.Oven_cell[36]:=FALSE;	
END_IF
IF CellMemory[CellNo.Oven_M37].Cell THEN
	P3User2_Par.Oven_cell[37]:=TRUE;
	ELSE
	P3User2_Par.Oven_cell[37]:=FALSE;	
END_IF

IF CellMemory[CellNo.Oven_M38].Cell THEN
	P3User2_Par.Oven_cell[38]:=TRUE;
	ELSE
	P3User2_Par.Oven_cell[38]:=FALSE;	
END_IF

IF CellMemory[CellNo.Oven_M39].Cell THEN
	P3User2_Par.Oven_cell[39]:=TRUE;
	ELSE
	P3User2_Par.Oven_cell[39]:=FALSE;	
END_IF
IF CellMemory[CellNo.Oven_M40].Cell THEN
	P3User2_Par.Oven_cell[40]:=TRUE;
	ELSE
	P3User2_Par.Oven_cell[40]:=FALSE;	
END_IF
IF CellMemory[CellNo.Oven_M41].Cell THEN
	P3User2_Par.Oven_cell[41]:=TRUE;
	ELSE
	P3User2_Par.Oven_cell[41]:=FALSE;	
END_IF
IF CellMemory[CellNo.Oven_M42].Cell THEN
	P3User2_Par.Oven_cell[42]:=TRUE;
	ELSE
	P3User2_Par.Oven_cell[42]:=FALSE;	
END_IF

